TYPE "LBP_typeNCVariableTokenDateAndTime"
TITLE = LBP_ReadVar and LBP_WriteVar Interface / Interface LBP_ReadVar et LBP_WriteVar
// User Data Type for LBP_ReadVar[FB2] and LBP_WriteVar[FB3] Parameters / Type de données utilisateur pour les paramètres LBP_ReadVar[FB2] et LBP_WriteVar[FB3]
   STRUCT
      token : "LBP_typeNCVariableToken";   // User Data Type for LBP_ReadVar[FB2] and LBP_WriteVar[FB3] Input Parameter Addrx / Type de données utilisateur pour les paramètres d'entrée Addrx LBP_ReadVar[FB2] et LBP_WriteVar[FB3]
      value : Date_And_Time;   // Data Type for LBP_ReadVar[FB2] and LBP_WriteVar[FB3] InOut Parameter SDx / Type de données pour les paramètres E/S SDx LBP_ReadVar[FB2] et LBP_WriteVar[FB3]
   END_STRUCT;
END_TYPE

TYPE "LBP_typeNCVariableTokenInt"
TITLE = LBP_ReadVar and LBP_WriteVar Interface / Interface LBP_ReadVar et LBP_WriteVar
// User Data Type for LBP_ReadVar[FB2] and LBP_WriteVar[FB3] Parameters / Type de données utilisateur pour les paramètres LBP_ReadVar[FB2] et LBP_WriteVar[FB3]
   STRUCT
      token : "LBP_typeNCVariableToken";   // User Data Type for LBP_ReadVar[FB2] and LBP_WriteVar[FB3] Input Parameter Addrx / Type de données utilisateur pour les paramètres d'entrée Addrx LBP_ReadVar[FB2] et LBP_WriteVar[FB3]
      value : Int;   // Data Type for LBP_ReadVar[FB2] and LBP_WriteVar[FB3] InOut Parameter SDx / Type de données pour les paramètres E/S SDx LBP_ReadVar[FB2] et LBP_WriteVar[FB3]
   END_STRUCT;
END_TYPE

TYPE "LBP_typeNCVariableTokenLReal"
TITLE = LBP_ReadVar and LBP_WriteVar Interface / Interface LBP_ReadVar et LBP_WriteVar
// User Data Type for LBP_ReadVar[FB2] and LBP_WriteVar[FB3] Parameters / Type de données utilisateur pour les paramètres LBP_ReadVar[FB2] et LBP_WriteVar[FB3]
   STRUCT
      token : "LBP_typeNCVariableToken";   // User Data Type for LBP_ReadVar[FB2] and LBP_WriteVar[FB3] Input Parameter Addrx / Type de données utilisateur pour les paramètres d'entrée Addrx LBP_ReadVar[FB2] et LBP_WriteVar[FB3]
      value : LReal;   // Data Type for LBP_ReadVar[FB2] and LBP_WriteVar[FB3] InOut Parameter SDx / Type de données pour les paramètres E/S SDx LBP_ReadVar[FB2] et LBP_WriteVar[FB3]
   END_STRUCT;
END_TYPE

TYPE "LBP_typeNCVariableTokenReal"
TITLE = LBP_ReadVar and LBP_WriteVar Interface / Interface LBP_ReadVar et LBP_WriteVar
// User Data Type for LBP_ReadVar[FB2] and LBP_WriteVar[FB3] Parameters / Type de données utilisateur pour les paramètres LBP_ReadVar[FB2] et LBP_WriteVar[FB3]
   STRUCT
      token : "LBP_typeNCVariableToken";   // User Data Type for LBP_ReadVar[FB2] and LBP_WriteVar[FB3] Input Parameter Addrx / Type de données utilisateur pour les paramètres d'entrée Addrx LBP_ReadVar[FB2] et LBP_WriteVar[FB3]
      value : Real;   // Data Type for LBP_ReadVar[FB2] and LBP_WriteVar[FB3] InOut Parameter SDx / Type de données pour les paramètres E/S SDx LBP_ReadVar[FB2] et LBP_WriteVar[FB3]
   END_STRUCT;
END_TYPE

TYPE "LBP_typeNCVariableTokenSInt"
TITLE = LBP_ReadVar and LBP_WriteVar Interface / Interface LBP_ReadVar et LBP_WriteVar
// User Data Type for LBP_ReadVar[FB2] and LBP_WriteVar[FB3] Parameters / Type de données utilisateur pour les paramètres LBP_ReadVar[FB2] et LBP_WriteVar[FB3]
   STRUCT
      token : "LBP_typeNCVariableToken";   // User Data Type for LBP_ReadVar[FB2] and LBP_WriteVar[FB3] Input Parameter Addrx / Type de données utilisateur pour les paramètres d'entrée Addrx LBP_ReadVar[FB2] et LBP_WriteVar[FB3]
      value : SInt;   // Data Type for LBP_ReadVar[FB2] and LBP_WriteVar[FB3] InOut Parameter SDx / Type de données pour les paramètres E/S SDx LBP_ReadVar[FB2] et LBP_WriteVar[FB3]
   END_STRUCT;
END_TYPE

TYPE "LBP_typeNCVariableTokenString"
TITLE = LBP_ReadVar and LBP_WriteVar Interface / Interface LBP_ReadVar et LBP_WriteVar
// User Data Type for LBP_ReadVar[FB2] and LBP_WriteVar[FB3] Parameters / Type de données utilisateur pour les paramètres LBP_ReadVar[FB2] et LBP_WriteVar[FB3]
   STRUCT
      token : "LBP_typeNCVariableToken";   // User Data Type for LBP_ReadVar[FB2] and LBP_WriteVar[FB3] Input Parameter Addrx / Type de données utilisateur pour les paramètres d'entrée Addrx LBP_ReadVar[FB2] et LBP_WriteVar[FB3]
      value : String;   // Data Type for LBP_ReadVar[FB2] and LBP_WriteVar[FB3] InOut Parameter SDx / Type de données pour les paramètres E/S SDx LBP_ReadVar[FB2] et LBP_WriteVar[FB3]
   END_STRUCT;
END_TYPE

TYPE "LBP_typeNCVariableTokenUDInt"
TITLE = LBP_ReadVar and LBP_WriteVar Interface / Interface LBP_ReadVar et LBP_WriteVar
// User Data Type for LBP_ReadVar[FB2] and LBP_WriteVar[FB3] Parameters / Type de données utilisateur pour les paramètres LBP_ReadVar[FB2] et LBP_WriteVar[FB3]
   STRUCT
      token : "LBP_typeNCVariableToken";   // User Data Type for LBP_ReadVar[FB2] and LBP_WriteVar[FB3] Input Parameter Addrx / Type de données utilisateur pour les paramètres d'entrée Addrx LBP_ReadVar[FB2] et LBP_WriteVar[FB3]
      value : UDInt;   // Data Type for LBP_ReadVar[FB2] and LBP_WriteVar[FB3] InOut Parameter SDx / Type de données pour les paramètres E/S SDx LBP_ReadVar[FB2] et LBP_WriteVar[FB3]
   END_STRUCT;
END_TYPE

TYPE "LBP_typeNCVariableTokenUInt"
TITLE = LBP_ReadVar and LBP_WriteVar Interface / Interface LBP_ReadVar et LBP_WriteVar
// User Data Type for LBP_ReadVar[FB2] and LBP_WriteVar[FB3] Parameters / Type de données utilisateur pour les paramètres LBP_ReadVar[FB2] et LBP_WriteVar[FB3]
   STRUCT
      token : "LBP_typeNCVariableToken";   // User Data Type for LBP_ReadVar[FB2] and LBP_WriteVar[FB3] Input Parameter Addrx / Type de données utilisateur pour les paramètres d'entrée Addrx LBP_ReadVar[FB2] et LBP_WriteVar[FB3]
      value : UInt;   // Data Type for LBP_ReadVar[FB2] and LBP_WriteVar[FB3] InOut Parameter SDx / Type de données pour les paramètres E/S SDx LBP_ReadVar[FB2] et LBP_WriteVar[FB3]
   END_STRUCT;
END_TYPE

TYPE "LBP_typeNCVariableTokenUSInt"
TITLE = LBP_ReadVar and LBP_WriteVar Interface / Interface LBP_ReadVar et LBP_WriteVar
// User Data Type for LBP_ReadVar[FB2] and LBP_WriteVar[FB3] Parameters / Type de données utilisateur pour les paramètres LBP_ReadVar[FB2] et LBP_WriteVar[FB3]
   STRUCT
      token : "LBP_typeNCVariableToken";   // User Data Type for LBP_ReadVar[FB2] and LBP_WriteVar[FB3] Input Parameter Addrx / Type de données utilisateur pour les paramètres d'entrée Addrx LBP_ReadVar[FB2] et LBP_WriteVar[FB3]
      value : USInt;   // Data Type for LBP_ReadVar[FB2] and LBP_WriteVar[FB3] InOut Parameter SDx / Type de données pour les paramètres E/S SDx LBP_ReadVar[FB2] et LBP_WriteVar[FB3]
   END_STRUCT;
END_TYPE

DATA_BLOCK "DB_WAF"   // DB12
{ S7_Optimized_Access := 'TRUE' }
// stored: MemoryReserve 100
   VAR
      bTest : Array[0..63] of Bool;
      bSpy : Array[0..63] of Bool;
      Sonplas : Struct
         OperateInOutCollision : Bool;
      END_STRUCT;
      BwLoader : Struct
         Safe : Bool;
         Auto : Bool;
      END_STRUCT;
      CtrlInEnable : Bool := true;
      CtrlOutEnable : Bool := true;
      CtrlBwEnable : Bool := true;
      U2States : Byte;
      ResetPartPosition : Bool;
      HMI_Pos : Bool;
      PLC_Pos : Bool;
      NewTag : Bool;
      NewTag_1 : Bool;
   END_VAR
BEGIN
END_DATA_BLOCK

DATA_BLOCK "DB_HMICmd"   // DB86
{ S7_Optimized_Access := 'TRUE' }
// stored: MemoryReserve 100
   VAR
      IntGateCloseReq : Bool;
      IntGateOpenReq : Bool;
      ExtGateCloseReq : Bool;
      ExtGateOpenReq : Bool;
      IntGateCloseCmd : Bool;
      IntGateOpenCmd : Bool;
      ExtGateCloseCmd : Bool;
      ExtGateOpenCmd : Bool;
      BlowingCmd : Bool;
   END_VAR
BEGIN
END_DATA_BLOCK

DATA_BLOCK "DB_HMISetting"   // DB1306
{ S7_Optimized_Access := 'FALSE' }
AUTHOR : DAT
NAME : IHM_SETT
// stored: AutoNumber false
   VAR RETAIN
      GasAssistSetPoint : Real;
      CoolingVentilatorSetpoint : Real;   // @Precision:0 @Unit:% @Min:0 @Max:100
      TemperatureCoolingSetpoint : Real;   // @Precision:1 @Unit:°C @Min:0 @Max:50
      BlowingSetpoint : Real;   // @Precision:0 @Unit:ms @Min:0 @Max:500
      WorkingMode : Struct
         EmptyingReq : Bool;
      END_STRUCT;
      Sonplas : Struct
         LimitMax : Real;
         LimitCtrlMax : Real;
         LimitCtrlMin : Real;
         LimitMin : Real;
         CorrectionMax : Real;
         CorrectionMin : Real;
      END_STRUCT;
      LockDoorReq : Bool;
      UnlockDoorReq : Bool;
      StartAutoReq : Bool;
      StopAutoReq : Bool;
      Shuttle1Enable : Bool;
      Shuttle2Enable : Bool;
   END_VAR
BEGIN
END_DATA_BLOCK

DATA_BLOCK "DB_HMIStatus"   // DB95
{ S7_Optimized_Access := 'TRUE' }
// stored: MemoryReserve 100
   VAR
      WarmUpOn : Bool := FALSE;
      WarmUpTime : Real := 30.0;
      KeyLaserOn : Bool := TRUE;
      Shutter_laser_closed : Bool := FALSE;
      Sonplas : Struct
         LastMeasure : Real;
         CurrentCorrection : Real;
         CouplerOk : Bool;
         Ready : Bool;
      END_STRUCT;
   END_VAR
BEGIN
END_DATA_BLOCK

DATA_BLOCK "DB_MachineOptions"   // DB1300
{ S7_Optimized_Access := 'FALSE'; DB_Accessible_From_OPC_UA := 'FALSE' }
// stored: AutoNumber false, DBAccessibleFromOPCUA false, DBAccessibleFromWebserver false
   VAR RETAIN
      UPSPresent : Bool;
      Fixture : Struct
         Passive_Open : Bool;
      END_STRUCT;
      Mach_MONO_DUO : Bool;
      Chiller : Struct
         Termotek : Bool := TRUE;
         SMC : Bool := FALSE;
      END_STRUCT;
   END_VAR
BEGIN
END_DATA_BLOCK

DATA_BLOCK "DB_PLC_ISO_IHM"   // DB1302
{ S7_Optimized_Access := 'FALSE' }
AUTHOR : SAN
FAMILY : DPR
NAME : HMI
// stored: AutoNumber false
   VAR RETAIN
      WarmUpOn : Bool := FALSE;   // Moved to DB_HMI_Status
      KeyLaserOn : Bool := TRUE;   // Moved to DB_HMI_Status
      KeySaveParameters : Bool := FALSE;   // Not used
      bStopAfterEmptying : Bool := FALSE;   // A VOIR SI ENCORE UTILE
      Chan1_running : Bool := TRUE;   // Moved to DB_HMI_Status
      Chan2_running : Bool := FALSE;   // Moved to DB_HMI_Status
      Chan3_running : Bool := FALSE;   // Moved to DB_HMI_Status
      Chan4_running : Bool := FALSE;   // Moved to DB_HMI_Status
      StopAtNextReq { S7_SetPoint := 'True'} : Bool := FALSE;   // Moved to DB_HMI_Status
      AllChanStop : Bool := FALSE;   // Moved to DB_HMI_Status
      LoaderAutomaticMode : Bool := FALSE;   // A VOIR SI ENCORE UTILE
      LoaderManualMode : Bool := TRUE;   // A VOIR SI ENCORE UTILE
      NoCameraPresent : Bool := FALSE;   // Not used
      PremeasureZexists : Bool := FALSE;   // Not used
      PremeasureCexists : Bool := FALSE;   // Not used
      PLCFunctNotFinished : Bool := FALSE;   // Not used
      StartChangePart_station1 : Bool := FALSE;   // A VOIR SI ENCORE UTILE
      StartCheckPart_fixture1 : Bool := FALSE;   // A VOIR SI ENCORE UTILE
      Loader1PartLoad : Bool := FALSE;   // A VOIR SI ENCORE UTILE
      Loader1PartUnload : Bool := FALSE;   // A VOIR SI ENCORE UTILE
      Loader1ShiftLoad : Bool := FALSE;   // A VOIR SI ENCORE UTILE
      Loader1ShiftUnload : Bool := FALSE;   // A VOIR SI ENCORE UTILE
      Loader1LoadOpened : Bool := TRUE;   // A VOIR SI ENCORE UTILE
      Loader1UnloadOpened : Bool := TRUE;   // A VOIR SI ENCORE UTILE
      PartOnFixture1 : Bool := FALSE;   // A VOIR SI ENCORE UTILE
      MasterOnFixture1 : Bool := FALSE;   // A VOIR SI ENCORE UTILE
      StartChangePart_station2 : Bool := FALSE;   // A VOIR SI ENCORE UTILE
      StartCheckPart_fixture2 : Bool := FALSE;   // A VOIR SI ENCORE UTILE
      Loader2PartLoad : Bool := FALSE;   // A VOIR SI ENCORE UTILE
      Loader2PartUnload : Bool := FALSE;   // A VOIR SI ENCORE UTILE
      Loader2ShiftLoad : Bool := FALSE;   // A VOIR SI ENCORE UTILE
      Loader2ShiftUnload : Bool := FALSE;   // A VOIR SI ENCORE UTILE
      Loader2LoadOpened : Bool := FALSE;   // A VOIR SI ENCORE UTILE
      Loader2UnloadOpened : Bool := FALSE;   // A VOIR SI ENCORE UTILE
      PartOnFixture2 : Bool := FALSE;   // A VOIR SI ENCORE UTILE
      MasterOnFixture2 : Bool := FALSE;   // A VOIR SI ENCORE UTILE
      StartChangePart_station3 : Bool := FALSE;   // A VOIR SI ENCORE UTILE
      StartCheckPart_fixture3 : Bool := FALSE;   // A VOIR SI ENCORE UTILE
      Loader3PartLoad : Bool := FALSE;   // A VOIR SI ENCORE UTILE
      Loader3PartUnload : Bool := FALSE;   // A VOIR SI ENCORE UTILE
      Loader3ShiftLoad : Bool := FALSE;   // A VOIR SI ENCORE UTILE
      Loader3ShiftUnload : Bool := FALSE;   // A VOIR SI ENCORE UTILE
      Loader3LoadOpened : Bool := FALSE;   // A VOIR SI ENCORE UTILE
      Loader3UnloadOpened : Bool := FALSE;   // A VOIR SI ENCORE UTILE
      PartOnFixture3 : Bool := FALSE;   // A VOIR SI ENCORE UTILE
      MasterOnFixture3 : Bool := FALSE;   // A VOIR SI ENCORE UTILE
      Part_KO_go_outside_mach : Bool := TRUE;   // Not used
      MasterOnMachine : Bool := FALSE;   // Not used
      Part_position_1 : Bool := FALSE;   // A VOIR COMMENT GERER AVEC TRACABILITY
      Part_position_2 : Bool := FALSE;   // A VOIR COMMENT GERER AVEC TRACABILITY
      Part_position_3 : Bool := FALSE;   // A VOIR COMMENT GERER AVEC TRACABILITY
      Part_position_4 : Bool := FALSE;   // A VOIR COMMENT GERER AVEC TRACABILITY
      Part_position_5 : Bool := FALSE;   // A VOIR COMMENT GERER AVEC TRACABILITY
      Part_position_6 : Bool := FALSE;   // A VOIR COMMENT GERER AVEC TRACABILITY
      Part_position_7 : Bool := FALSE;   // A VOIR COMMENT GERER AVEC TRACABILITY
      Part_position_8 : Bool := FALSE;   // A VOIR COMMENT GERER AVEC TRACABILITY
      Part_position_9 : Bool := FALSE;   // A VOIR COMMENT GERER AVEC TRACABILITY
      Part_position_10 : Bool := FALSE;   // A VOIR COMMENT GERER AVEC TRACABILITY
      Part_position_11 : Bool := FALSE;   // A VOIR COMMENT GERER AVEC TRACABILITY
      Part_position_12 : Bool := FALSE;   // A VOIR COMMENT GERER AVEC TRACABILITY
      Part_position_13 : Bool := FALSE;   // A VOIR COMMENT GERER AVEC TRACABILITY
      Part_position_14 : Bool := FALSE;   // A VOIR COMMENT GERER AVEC TRACABILITY
      Part_position_15 : Bool := FALSE;   // A VOIR COMMENT GERER AVEC TRACABILITY
      Part_position_16 : Bool := FALSE;   // A VOIR COMMENT GERER AVEC TRACABILITY
      WarmUpTime : Int := 30;   // Moved to DB_HMI_Status
      Stop_For_BackWall_Wear_1 : Bool := FALSE;   // Moved to DB_HMI_Status
      Stop_For_BackWall_Wear_2 : Bool := FALSE;   // Moved to DB_HMI_Status
      Cleaning_Station_1 : Bool := FALSE;   // Moved to DB_HMI_Status
      Cleaning_Station_2 : Bool := FALSE;   // Moved to DB_HMI_Status
      Cleaning_Backwall_1 : Bool := FALSE;   // Moved to DB_HMI_Status
      Cleaning_Backwall_2 : Bool := FALSE;   // Moved to DB_HMI_Status
      Shutter_laser_closed : Bool := FALSE;   // Moved to DB_HMI_Status
      Pressure_Stop_Machine : Bool := FALSE;   // Moved to DB_HMI_Status
      Set_Bad_Part_On_Fixture : Bool := FALSE;   // Moved to DB_HMI_Status
      Reserve12 : Bool := FALSE;   // Not used
      Reserve13 : Bool := FALSE;   // Not used
      Reserve14 : Bool := FALSE;   // Not used
      Reserve15 : Bool := FALSE;   // Not used
      SemiAuto_RunEmpty : Bool := FALSE;   // A VOIR SI ENCORE UTILE
      "SemiAuto_Unload_C-Fixture" : Bool := FALSE;   // A VOIR SI ENCORE UTILE
      Reserve18 : Bool := FALSE;   // Not used
      Cnt_Washing_Loader_1 : Int := 1;   // A VOIR SI ENCORE UTILE
      Cnt_Washing_Loader_2 : Int := 0;   // A VOIR SI ENCORE UTILE
      Cnt_Part_Backwall_1 : Int := 16;   // Moved to DB_HMI_Status
      Cnt_Part_Backwall_2 : Int := 0;   // Moved to DB_HMI_Status
      Cnt_Part_Wash_Backwall_1 : Int := 26;   // Moved to DB_HMI_Status
      Cnt_Part_Wash_Backwall_2 : Int := 0;   // Moved to DB_HMI_Status
      Cnt_Part_Blow_Fixture_1 : Int;   // Moved to DB_HMI_Status
      Cnt_Part_Blow_Fixture_2 : Int;   // Moved to DB_HMI_Status
      Setpoint_laser_air_process : Real;   // Not used
      StopMachine : Bool;   // Not used
      BadPartOnFixture : Bool;   // Not used
   END_VAR
BEGIN
END_DATA_BLOCK

DATA_BLOCK "DB_LoaderOptions"   // DB1305
{ S7_Optimized_Access := 'TRUE' }
AUTHOR : SAN
// stored: AutoNumber false, IsRetainMemResEnabled true, MemoryReserve 20, RetainMemoryReserve 20
   VAR RETAIN
      ExtLoadUnload : Struct
         SeparatePos : Bool;
         CommonPos : Bool;
         Disabled : Bool;
      END_STRUCT;
      Blowing : Struct
         Inside : Bool;
         NearSas : Bool;
         Disabled : Bool;
      END_STRUCT;
      Washing : Struct
         Enabled : Bool;
         Disabled : Bool;
      END_STRUCT;
      PartControl : Struct
         Individual : Bool;
         Common : Bool;
         Disabled : Bool;
         AnalogMeasure : Bool;
         DigitalMeasure : Bool;
      END_STRUCT;
   END_VAR
   VAR
      Stop_Restart : Struct
         BasicVersion : Bool;
      END_STRUCT;
      IntLoadUnload : Struct
         SeparatePos : Bool;
         CommonPos : Bool;
      END_STRUCT;
      BwLoadUnload : Struct
         SeparatePos : Bool;
         CommonPos : Bool;
      END_STRUCT;
      BwControl : Struct
         UndrilledDrilledCtrlSeparate : Bool;
         UndrilledDrilledCtrlCommon : Bool;
         Disabled : Bool;
      END_STRUCT;
      ActPartControlIn : Struct
         Stop : Bool := TRUE;
      END_STRUCT;
      ActPartControlOut : Struct
         Stop : Bool := TRUE;
      END_STRUCT;
      ActBwControlIn : Struct
         Stop : Bool := TRUE;
      END_STRUCT;
      Fixture : Struct
         UnloadingDisabled : Bool;
         LoadingDisabled : Bool;
         BlowingDisabled : Bool;
         ReleaseDisabled : Bool;
         V_InitDisabled : Bool;
         W_InitDisabled : Bool;
      END_STRUCT;
   END_VAR
BEGIN
END_DATA_BLOCK

DATA_BLOCK "DB_ActiveAlarms"   // DB115
{ S7_Optimized_Access := 'TRUE' }
// stored: MemoryReserve 100
   VAR
      NumberOfActiveAlarms : DInt;
      ActiveAlarms : Array[0..50] of "UDT_Alarms";
      Update { S7_SetPoint := 'True'} : Byte;   // A modifier lors d'un Acknowledge
   END_VAR
BEGIN
END_DATA_BLOCK

DATA_BLOCK "DB_FormatMsg"   // DB18
{ S7_Optimized_Access := 'TRUE' }
// stored: MemoryReserve 100
   VAR
      Msg : Array[0..863] of "UDT_FormatMsg";
   END_VAR
BEGIN
END_DATA_BLOCK

DATA_BLOCK "DB_AxisPosMachineNC"   // DB82
{ S7_Optimized_Access := 'TRUE' }
// stored: MemoryReserve 100
   VAR
      Axis_X : Struct
         Load : LReal := 249.3;
         Unload : LReal := 324.5;
         Blowing : LReal := 287.3;
      END_STRUCT;
      Axis_Y : Struct
         Load : LReal := 55.02;
         Unload : LReal := 55.02;
         Blowing : LReal := 55.02;
      END_STRUCT;
      Axis_B : Struct
         Load : LReal := 0.0;
         Unload : LReal := 0.0;
         Blowing : LReal := 0.0;
      END_STRUCT;
      Axis_ZM : Struct
         Safe : Real := 145.0;
      END_STRUCT;
      Axis_ZL : Struct
         Safe : Real := 14.0;
      END_STRUCT;
   END_VAR
BEGIN
END_DATA_BLOCK

DATA_BLOCK "DB_AxisPosMachinePLC"   // DB103
{ S7_Optimized_Access := 'TRUE' }
// stored: AutoNumber false, MemoryReserve 100
   VAR
      Axis_U1 : Struct
         ExtLoadUnloadAuto : LReal := -3370.0;
         ExtLoadUnloadManu : LReal := -3365.0;
         PartControl : LReal := -3257.0;
         BwLoad : LReal := -1886.83;
         BwUnLoad : LReal := -1962.83;
         BwControl : LReal := -1775.0;
         IntLoadUnload : LReal := -0.2;
         ExtGateExt : LReal := -1164.0;
         IntGateExt : LReal := -857.0;
         ExtGateInt : LReal := -809.0;
         IntGateInt : LReal := -502.0;
         Sas : LReal := -833.0;
         Blowing : LReal := 36.0;
         IntLoadUnloadOP : LReal := 76.0;
      END_STRUCT;
      Axis_U2 : Struct
         ExtLoadUnloadAuto : LReal := -3370.0;
         ExtLoadUnloadManu : LReal := -3365.0;
         PartControl : LReal := -3257.0;
         BwLoad : LReal := -1886.78;
         BwUnLoad : LReal := -1962.78;
         BwControl : LReal := -1775.0;
         IntLoadUnload : LReal := -0.11;
         ExtGateExt : LReal := -1164.0;
         IntGateExt { ExternalAccessible := 'False'; ExternalVisible := 'False'; ExternalWritable := 'False'} : LReal := -857.0;
         ExtGateInt : LReal := -809.0;
         IntGateInt : LReal := -502.0;
         Sas : LReal := -833.0;
         Blowing : LReal := 36.0;
         IntLoadUnloadOP : LReal := 76.0;
      END_STRUCT;
      Axis_V : Struct
         Shuttle_1 : Struct
            LoadUnload : LReal := 17.95;
            Blowing : LReal := 17.95;
         END_STRUCT;
         Shuttle_2 : Struct
            LoadUnload : LReal := -0.48;
            Blowing : LReal := -0.48;
         END_STRUCT;
         Safe : LReal := -0.48;
         Fixture : Struct
            Safe : LReal := 40.0;
            Load : LReal := 192.62;   // 193.52
            Unload : LReal := 192.62;   // 193.52
            Blowing : LReal := 192.62;   // 193.52
         END_STRUCT;
      END_STRUCT;
      Axis_W : Struct
         Shuttle_1 : Struct
            Approach : LReal := -17.61;
            LoadUnload : LReal := -19.61;
            Blowing : LReal := -5.0;
         END_STRUCT;
         Shuttle_2 : Struct
            Approach : LReal := -17.81;
            LoadUnload : LReal := -19.81;
            Blowing : LReal := -5.0;
         END_STRUCT;
         Safe : LReal := 28.5;
         Fixture : Struct
            Safe : LReal := 28.5;
            Load : LReal := -0.8;
            Blowing : LReal := 15.0;
            Unload : LReal := -0.9;
            Approach : LReal := 2.0;
         END_STRUCT;
      END_STRUCT;
   END_VAR
BEGIN
END_DATA_BLOCK

DATA_BLOCK "DB_DataFinalPart"   // DB700
{ S7_Optimized_Access := 'TRUE' }
// stored: AutoNumber false, MemoryReserve 100
   VAR
      FinalPart : Array[0..100] of "UDT_Tracability";
   END_VAR
BEGIN
END_DATA_BLOCK

DATA_BLOCK "DB_DataPositions"   // DB701
{ S7_Optimized_Access := 'TRUE' }
// stored: AutoNumber false, MemoryReserve 100
   VAR
      Position : Array[0..52] of "UDT_Tracability";
   END_VAR
BEGIN
END_DATA_BLOCK

DATA_BLOCK "DB_OPC_Buttons"   // DB92
{ S7_Optimized_Access := 'TRUE' }
// stored: MemoryReserve 100
   VAR
      Door : "UDT_OPC_Button";
      Empty : "UDT_OPC_Button";
      Start : "UDT_OPC_Button";
      Stop : "UDT_OPC_Button";
      Powermeter { S7_SetPoint := 'True'} : "UDT_OPC_Button";
      GasAssist { S7_SetPoint := 'True'} : "UDT_OPC_Button";
      GripperUndrilledClamp : Struct
         Close : "UDT_OPC_Button";
         Open { S7_SetPoint := 'True'} : "UDT_OPC_Button";
         IsClosed { S7_SetPoint := 'True'} : Bool;
         IsOpened { S7_SetPoint := 'True'} : Bool;
      END_STRUCT;
      GripperDrilledClamp : Struct
         Close : "UDT_OPC_Button";
         Open { S7_SetPoint := 'True'} : "UDT_OPC_Button";
         IsClosed { S7_SetPoint := 'True'} : Bool;
         IsOpened { S7_SetPoint := 'True'} : Bool;
      END_STRUCT;
      SITestStop { S7_SetPoint := 'True'} : "UDT_OPC_Button";
      FixtureClamp { S7_SetPoint := 'True'} : "UDT_OPC_Button";
      FixtureVacuum { S7_SetPoint := 'True'} : "UDT_OPC_Button";
      Aspiration { S7_SetPoint := 'True'} : "UDT_OPC_Button";
      LoaderAuto { S7_SetPoint := 'True'} : "UDT_OPC_Button";
      LoaderSemiAuto { S7_SetPoint := 'True'} : "UDT_OPC_Button";
      Backlight { S7_SetPoint := 'True'} : "UDT_OPC_Button";
      ObservationCamera { S7_SetPoint := 'True'} : "UDT_OPC_Button";
      MainDoor { S7_SetPoint := 'True'} : "UDT_OPC_Button";
      WarmUp { S7_SetPoint := 'True'} : "UDT_OPC_Button";
      MachineLight { S7_SetPoint := 'True'} : "UDT_OPC_Button";
   END_VAR
BEGIN
END_DATA_BLOCK

DATA_BLOCK "DB_OPC_Axis"   // DB102
{ S7_Optimized_Access := 'TRUE' }
// stored: MemoryReserve 100
   VAR
      ActualValues : Struct
         NumberOfAxes { S7_SetPoint := 'True'} : DInt;
         Axes : Array[0..100] of "UDT_OPC_ActualValuesAxis";
      END_STRUCT;
      TaughtPositions : Struct
         NumberOfItems { S7_SetPoint := 'True'} : DInt;
         Items : Array[0..100] of "UDT_OPC_TaughtPositionsItems";
      END_STRUCT;
      Teach : Struct
         Buttons : Struct
            Teach : "UDT_OPCButtons";
         END_STRUCT;
         Parameters : Struct
            AxisId : DInt;
            PositionId : DInt;
         END_STRUCT;
         Current : Struct
            ActualPosition : LReal;
            TaughtPosition : LReal;
         END_STRUCT;
      END_STRUCT;
   END_VAR
BEGIN
END_DATA_BLOCK

DATA_BLOCK "DB_OPC_Machine"   // DB15
{ S7_Optimized_Access := 'TRUE' }
// stored: MemoryReserve 100
   VAR
      Parts : Struct
         Out : Struct
            Station1 : Struct
               LoaderDrilled : SInt;
               LoaderUndrilled : SInt;
               ShuttleDrilled : SInt;
               ShuttleUndrilled : SInt;
               WorkClamp : SInt;
            END_STRUCT;
         END_STRUCT;
      END_STRUCT;
      State : Struct
         Current : Struct
            CanLockDoor : Bool;
            CanUnlockDoor : Bool;
            CncMode : Byte;
            LoadingMode : Byte;
            IsDoorLocked : Bool;
            IsEmptying : Bool;
            IsInitialized : Bool;
            IsRunning : Bool;
            MachineOverride : Byte;
         END_STRUCT;
         Requests : Struct
            LoadingMode : Struct
               RequestChangeMode : Bool;
               TargetMode : Byte;
            END_STRUCT;
            RequestLockDoor : Bool;
            RequestStartAuto : Bool;
            RequestStartEmptying : Bool;
            RequestStopAuto : Bool;
            RequestStopEmptying : Bool;
            RequestUnlockDoor : Bool;
         END_STRUCT;
      END_STRUCT;
   END_VAR
   VAR RETAIN
      Parameters : Struct
         GasAssistSetPoint : Real;
         CoolingVentilatorSetpoint : Real;
         TemperatureCoolingSetpoint : Real;
         BlowingSetpoint : Real;
         Shuttle1Enable : "UDT_BoolEnable";
         Shuttle2Enable { S7_SetPoint := 'True'} : "UDT_BoolEnable";
         ConsecutiveBwIn { S7_SetPoint := 'True'} : Int;
         Sequence : Struct
            Shuttle1 : Struct
               Main : Int;
               ShuttleInt : Int;
               ShuttleExt : Int;
               ControlIn : Int;
               ControlOut : Int;
               Blowing : Int;
               IntLoadUnload : Int;
               ExtLoadUnload : Int;
               BwLoadUnload : Int;
               BwControlIn : Int;
               ActControlIn : Int;
               ActControlOut : Int;
               ActBwControlIn : Int;
            END_STRUCT;
            Shuttle2 : Struct
               Main : Int;
               ShuttleInt : Int;
               ShuttleExt : Int;
               ControlIn : Int;
               ControlOut : Int;
               Blowing : Int;
               IntLoadUnload : Int;
               ExtLoadUnload : Int;
               BwLoadUnload : Int;
               BwControlIn : Int;
               ActControlIn : Int;
               ActControlOut : Int;
               ActBwControlIn : Int;
            END_STRUCT;
            Fixture : Struct
               Blowing : Int;
               Loading : Int;
               Unloading : Int;
               V_Init : Int;
               W_Init : Int;
            END_STRUCT;
         END_STRUCT;
         Presence : Struct
            Shuttle1UndrilledPart : Bool;
            Shuttle1UndrilledBw : Bool;
            Shuttle1DrilledPart : Bool;
            Shuttle1DrilledBw : Bool;
            Shuttle2UndrilledPart : Bool;
            Shuttle2UndrilledBw : Bool;
            Shuttle2DrilledPart : Bool;
            Shuttle2DrilledBw : Bool;
            GripperUndrilledPart : Bool;
            GripperUndrilledBw : Bool;
            GripperDrilledPart : Bool;
            GripperDrilledBw : Bool;
            FixtureUndrilledPart : Bool;
            FixtureUndrilledBw : Bool;
            FixtureDrilledPart : Bool;
            FixtureDrilledBw : Bool;
         END_STRUCT;
      END_STRUCT;
   END_VAR
BEGIN
END_DATA_BLOCK

DATA_BLOCK "DB_OPC_Alarms"   // DB117
{ S7_Optimized_Access := 'TRUE' }
// stored: MemoryReserve 100
   VAR
      NumberOfActiveAlarms : DInt;
      ActiveAlarms : Array[0..50] of "UDT_Alarms";
      Update { S7_SetPoint := 'True'} : Byte;   // A modifier lors d'un Acknowledge
   END_VAR
BEGIN
END_DATA_BLOCK

DATA_BLOCK "DB_BwLoaderExchange"   // DB101
{ S7_Optimized_Access := 'TRUE' }
// stored: MemoryReserve 100
   VAR
      Inputs : Struct
         LifeFlag : Int;
         JobDone : Bool;
         LockShuttle : Bool;
         DataSend : Int;
         DataReceive : Int;
         NoEmergencyStopAtBwLoader : Bool;
         SafetyDoorsClosedAtBwLoader : Bool;
         BwInErrorState : Int;
         UndrilledPartControl : Bool;
         DrilledPartControl : Bool;
         BackwallControl : Bool;
         BwLoaderInSafePos : Bool;
      END_STRUCT;
      Outputs : Struct
         LifeFlag : Int;
         LoaderRequest : Bool;
         LockShuttle : Bool;
         DataSend : Int;
         DataReceive : Int;
         NoEmergencyStopAtFemto : Bool;
         SafetyDoorsClosedAtFemto : Bool;
         FemtoInErrorState : Int;
         AutoMode : Bool;
         JogMode : Bool;
         GotoSafePos : Bool;
         Emptying : Bool;
         BW_CtrlInProgress : Bool;
      END_STRUCT;
   END_VAR
BEGIN
END_DATA_BLOCK

DATA_BLOCK "DB_OPC_RealTime"   // DB104
{ S7_Optimized_Access := 'TRUE' }
// stored: MemoryReserve 100
   VAR
      GripperUndrilledClampOpen : Bool;   // Test
      GripperUndrilledClampClosed : Bool;   // Test
      FixturePosition : Real;   // Test
      X_AxisBrakePressCtrl : Bool;   // Digital Input
      Y_AxisBrakePressCtrl : Bool;   // Digital Input
      BreakerCtrl : Bool;   // Digital Input
      CabinetTemperatureCtrl : Bool;   // Digital Input
      UpsPowerFailure : Bool;   // Digital Input
      AirPressureCtrl : Bool;   // Digital Input
      ShutterClosed : Bool;   // Digital Input
      AirDryerOK : Bool;   // Digital Input
      UPS_BatteryOK : Bool;   // Digital Input
      FrontDoorClosed : Bool;   // Digital Input
      InfeedReadyOkStart : Bool;   // Digital Input
      CoolingOK : Bool;   // Digital Input
      PowerReady : Bool;   // Digital Input
      AlarmI2T : Bool;   // Digital Input
      HeadLaserBusy : Bool;   // Digital Input
      HeadLaserBreaker : Bool;   // Digital Input
      FrontDoorLocked : Bool;   // Digital Input
      UPS_CommonAlarm : Bool;   // Digital Input
      UPS_BatteryLow : Bool;   // Digital Input
      HeadChillerHighPressure : Bool;   // Digital Input
      HeadChillerWaterTemperature : Bool;   // Digital Input
      HeadChillerFlow : Bool;   // Digital Input
      HeadChillerCollectivFault : Bool;   // Digital Input
      HeadChillerWaterLevel : Bool;   // Digital Input
      UpsByPassActive : Bool;   // Digital Input
      HeadChillerAmbiantTemperature : Bool;   // Digital Input
      LoadClampOpened : Bool;   // Digital Input
      LoadClampNotClosedWithPart : Bool;   // Digital Input
      UnloadClampOpened : Bool;   // Digital Input
      UpsFault : Bool;   // Digital Input
      InternalGateLocked : Bool;   // Digital Input
      ExternalGateLocked : Bool;   // Digital Input
      InverterActive : Bool;   // Digital Input
      UnloadClampNotClosedWithPart : Bool;   // Digital Input
      InternalGateOpened : Bool;   // Digital Input
      ExternalGateOpened : Bool;   // Digital Input
      PowerMeterBackCtrl : Bool;   // Digital Input
      PowerMeterFrontCtrl : Bool;   // Digital Input
      HeadChillerCutOff : Bool;   // Digital Input
      HeadChillerTemperature : Bool;   // Digital Input
      ClampingOpenCtrl : Bool;   // Digital Input
      B_AxisBrakeReleasedCtrl : Bool;   // Digital Input
      B_AxisReferencePoint : Bool;   // Digital Input
      SourceChillerHighPressure : Bool;   // Digital Input
      SourceChillerWaterTemperature : Bool;   // Digital Input
      SourceChillerFlow : Bool;   // Digital Input
      SourceChillerCollectivFault : Bool;   // Digital Input
      SourceChillerWaterLevel : Bool;   // Digital Input
      SourceChillerAmbiantTemperature : Bool;   // Digital Input
      SourceChillerCutOff : Bool;   // Digital Input
      SourceChillerTemperature : Bool;   // Digital Input
      OperatingCounter : Bool;   // Digital Output
      GeneralAirValve : Bool;   // Digital Output
      SmartLineDisable : Bool;   // Digital Output
      MachineLight : Bool;   // Digital Output
      MachineLightBack : Bool;   // Digital Output
      LightTowerOrange : Bool;   // Digital Output
      LightTowerRed : Bool;   // Digital Output
      LightTowerBlue : Bool;   // Digital Output
      LightTowerGreen : Bool;   // Digital Output
      LightTowerWhite : Bool;   // Digital Output
      Backlight : Bool;   // Digital Output
      InfeedON : Bool;   // Digital Output
      AxisActivation : Bool;   // Digital Output
      BuzzerActivation : Bool;   // Digital Output
      ElbaronPowerON : Bool;   // Digital Output
      ObservationCameraLight : Bool;   // Digital Output
      LaserExternalDoorOpening : Bool;   // Digital Output
      CoolingStart : Bool;   // Digital Output
      X_AxisBrakeActivation : Bool;   // Digital Output
      Y_AxisBrakeActivation : Bool;   // Digital Output
      AxisB_TeachInClampingPart : Bool;   // Digital Output
      EPO_UPS : Bool;   // Digital Output
      HeadLaserStart : Bool;   // Digital Output
      HeadLaserStop : Bool;   // Digital Output
      Axis2_PowerContactor : Bool;   // Digital Output
      GasAssistOn : Bool;   // Digital Output
      SmartLineReset : Bool;   // Digital Output
      XY_AxisPowerContactor : Bool;   // Digital Output
      LaserAirPressureProcess : Bool;   // Digital Output
      Bus60V_PowerContactor : Bool;   // Digital Output
      LoadClampClosing : Bool;   // Digital Output
      LoadClampOpening : Bool;   // Digital Output
      UnloadClampClosing : Bool;   // Digital Output
      UnloadClampOpening : Bool;   // Digital Output
      ClampingOpening : Bool;   // Digital Output
      ClampingClosing : Bool;   // Digital Output
      B_AxisBrakeRelease : Bool;   // Digital Output
      Suction : Bool;   // Digital Output
      ExternalGateClosing : Bool;   // Digital Output
      ExternalGateOpening : Bool;   // Digital Output
      InternalGateClosing : Bool;   // Digital Output
      InternalGateOpening : Bool;   // Digital Output
      PowerMeterRetract : Bool;   // Digital Output
      PowerMeterAdvance : Bool;   // Digital Output
      Blowing : Bool;   // Digital Output
      LaserPowerMeter : Real;   // Analog Input
      AxisB_ClampingPart : Real;   // Analog Input
      LaserAirPressureProcess_1 : Real;   // Analog Input
      InletAirPressure : Real;   // Analog Input
      AmbiantTemperature : Real;   // Analog Input
      MachineTemperature : Real;   // Analog Input
      Cold_WaterTemperatureInput { ExternalWritable := 'False'} : Real;   // Analog Input
      Cold_WaterTemperatureOutput : Real;   // Analog Input
      X_AxisTemperaturePT1000 : Real;   // Analog Input
      Y_AxisTemperaturePT1000 : Real;   // Analog Input
      X_AxisTemperaturePTC : Real;   // Analog Input
      Y_AxisTemperaturePTC : Real;   // Analog Input
      NozzleOverpressure : Real;   // Analog Input
      OpticalPathOverpressure : Real;   // Analog Input
      LaserHeadOverpressure : Real;   // Analog Input
      ZLAxisOverpressure : Real;   // Analog Input
      XYAxisOverpressure : Real;   // Analog Input
      LeftAspiration : Real;   // Analog Input
      RightAspiration : Real;   // Analog Input
      ClimTemperature : Real;   // Analog Input
      SensorControllerStation1 : Real;   // Analog Input
      CabinetTemperature : Real;   // Analog Input
      NozzleOverpressureSetPoint : Real;   // Analog Output
      VentilatorSetPoint : Real;   // Analog Output
      PropValveClimSetPoint : Real;   // Analog Output
   END_VAR
BEGIN
END_DATA_BLOCK

DATA_BLOCK "DB_OPC_AnalogInputs"   // DB83
{ S7_Optimized_Access := 'TRUE' }
// stored: MemoryReserve 100
   VAR
      NumberOfSignals : Int := 22;
      Parameters : Struct
         Delay : LReal;
         DiffErrorMax : LReal;
         DiffErrorMin : LReal;
         DiffWarnMax : LReal;
         DiffWarnMin : LReal;
         Id : DInt;
         ItemNumber : DInt;
         Offset : LReal := 1.0;
         Gain : LReal;
         Target : LReal;
      END_STRUCT;
      Signals : Array[0..100] of "UDT_OPC_Analog";
      Update { S7_SetPoint := 'True'} : Bool;
   END_VAR
BEGIN
   // Signals[1].DiffErrorMax : Unit:W
   // Signals[3].DiffErrorMax : Unit:bar
   // Signals[4].DiffErrorMax : Unit:°C
   // Signals[5].DiffErrorMax : Unit:°C
   // Signals[6].DiffErrorMax : Unit:°C
   // Signals[7].DiffErrorMax : Unit:°C
   // Signals[8].DiffErrorMax : Unit:°C
   // Signals[9].DiffErrorMax : Unit:°C
   // Signals[10].DiffErrorMax : Unit:°C
   // Signals[13].DiffErrorMax : Unit:bar
   // Signals[14].DiffErrorMax : Unit:bar
   // Signals[15].DiffErrorMax : Unit:bar
   // Signals[16].DiffErrorMax : Unit:bar
   // Signals[17].DiffErrorMax : Unit:bar
   // Signals[18].DiffErrorMax : Unit:mm/s
   // Signals[19].DiffErrorMax : Unit:mm/s
   // Signals[21].DiffErrorMax : Unit:°C
   // Signals[26].DiffErrorMax : Unit:°C
   // Signals[1].DiffErrorMin : Unit:W
   // Signals[3].DiffErrorMin : Unit:bar
   // Signals[4].DiffErrorMin : Unit:°C
   // Signals[5].DiffErrorMin : Unit:°C
   // Signals[6].DiffErrorMin : Unit:°C
   // Signals[7].DiffErrorMin : Unit:°C
   // Signals[8].DiffErrorMin : Unit:°C
   // Signals[9].DiffErrorMin : Unit:°C
   // Signals[10].DiffErrorMin : Unit:°C
   // Signals[13].DiffErrorMin : Unit:bar
   // Signals[14].DiffErrorMin : Unit:bar
   // Signals[15].DiffErrorMin : Unit:bar
   // Signals[16].DiffErrorMin : Unit:bar
   // Signals[17].DiffErrorMin : Unit:bar
   // Signals[18].DiffErrorMin : Unit:mm/s
   // Signals[19].DiffErrorMin : Unit:mm/s
   // Signals[21].DiffErrorMin : Unit:°C
   // Signals[26].DiffErrorMin : Unit:°C
   // Signals[1].DiffWarnMax : Unit:W
   // Signals[3].DiffWarnMax : Unit:bar
   // Signals[4].DiffWarnMax : Unit:°C
   // Signals[5].DiffWarnMax : Unit:°C
   // Signals[6].DiffWarnMax : Unit:°C
   // Signals[7].DiffWarnMax : Unit:°C
   // Signals[8].DiffWarnMax : Unit:°C
   // Signals[9].DiffWarnMax : Unit:°C
   // Signals[10].DiffWarnMax : Unit:°C
   // Signals[13].DiffWarnMax : Unit:bar
   // Signals[14].DiffWarnMax : Unit:bar
   // Signals[15].DiffWarnMax : Unit:bar
   // Signals[16].DiffWarnMax : Unit:bar
   // Signals[17].DiffWarnMax : Unit:bar
   // Signals[18].DiffWarnMax : Unit:mm/s
   // Signals[19].DiffWarnMax : Unit:mm/s
   // Signals[21].DiffWarnMax : Unit:°C
   // Signals[26].DiffWarnMax : Unit:°C
   // Signals[1].DiffWarnMin : Unit:W
   // Signals[3].DiffWarnMin : Unit:bar
   // Signals[4].DiffWarnMin : Unit:°C
   // Signals[5].DiffWarnMin : Unit:°C
   // Signals[6].DiffWarnMin : Unit:°C
   // Signals[7].DiffWarnMin : Unit:°C
   // Signals[8].DiffWarnMin : Unit:°C
   // Signals[9].DiffWarnMin : Unit:°C
   // Signals[10].DiffWarnMin : Unit:°C
   // Signals[13].DiffWarnMin : Unit:bar
   // Signals[14].DiffWarnMin : Unit:bar
   // Signals[15].DiffWarnMin : Unit:bar
   // Signals[16].DiffWarnMin : Unit:bar
   // Signals[17].DiffWarnMin : Unit:bar
   // Signals[18].DiffWarnMin : Unit:mm/s
   // Signals[19].DiffWarnMin : Unit:mm/s
   // Signals[21].DiffWarnMin : Unit:°C
   // Signals[26].DiffWarnMin : Unit:°C
   // Signals[1].Offset : Unit:W
   // Signals[3].Offset : Unit:bar
   // Signals[4].Offset : Unit:°C
   // Signals[5].Offset : Unit:°C
   // Signals[6].Offset : Unit:°C
   // Signals[7].Offset : Unit:°C
   // Signals[8].Offset : Unit:°C
   // Signals[9].Offset : Unit:°C
   // Signals[10].Offset : Unit:°C
   // Signals[13].Offset : Unit:bar
   // Signals[14].Offset : Unit:bar
   // Signals[15].Offset : Unit:bar
   // Signals[16].Offset : Unit:bar
   // Signals[17].Offset : Unit:bar
   // Signals[18].Offset : Unit:mm/s
   // Signals[19].Offset : Unit:mm/s
   // Signals[21].Offset : Unit:°C
   // Signals[26].Offset : Unit:°C
   // Signals[1].Target : Unit:W
   // Signals[3].Target : Unit:bar
   // Signals[4].Target : Unit:°C
   // Signals[5].Target : Unit:°C
   // Signals[6].Target : Unit:°C
   // Signals[7].Target : Unit:°C
   // Signals[8].Target : Unit:°C
   // Signals[9].Target : Unit:°C
   // Signals[10].Target : Unit:°C
   // Signals[13].Target : Unit:bar
   // Signals[14].Target : Unit:bar
   // Signals[15].Target : Unit:bar
   // Signals[16].Target : Unit:bar
   // Signals[17].Target : Unit:bar
   // Signals[18].Target : Unit:mm/s
   // Signals[19].Target : Unit:mm/s
   // Signals[21].Target : Unit:°C
   // Signals[26].Target : Unit:°C
   // Signals[1].Value : Unit:W
   // Signals[3].Value : Unit:bar
   // Signals[4].Value : Unit:°C
   // Signals[5].Value : Unit:°C
   // Signals[6].Value : Unit:°C
   // Signals[7].Value : Unit:°C
   // Signals[8].Value : Unit:°C
   // Signals[9].Value : Unit:°C
   // Signals[10].Value : Unit:°C
   // Signals[13].Value : Unit:bar
   // Signals[14].Value : Unit:bar
   // Signals[15].Value : Unit:bar
   // Signals[16].Value : Unit:bar
   // Signals[17].Value : Unit:bar
   // Signals[18].Value : Unit:mm/s
   // Signals[19].Value : Unit:mm/s
   // Signals[21].Value : Unit:°C
   // Signals[26].Value : Unit:°C
END_DATA_BLOCK

DATA_BLOCK "DB_OPC_Components"   // DB118
{ S7_Optimized_Access := 'TRUE' }
// stored: MemoryReserve 100
   VAR
      Backwalls : Struct
         LoaderDrilled : Byte;
         LoaderUndrilled : Byte;
         Shuttle2Drilled : Byte;
         Shuttle2Undrilled : Byte;
         ShuttleDrilled : Byte;
         ShuttleUndrilled : Byte;
         WorkClamp : Byte;
      END_STRUCT;
      Parts : Struct
         LoaderDrilled : Byte;
         LoaderUndrilled : Byte;
         Shuttle2Drilled : Byte;
         Shuttle2Undrilled : Byte;
         ShuttleDrilled : Byte;
         ShuttleUndrilled : Byte;
         WorkClamp : Byte;
      END_STRUCT;
      Update : Byte;
   END_VAR
BEGIN
END_DATA_BLOCK

DATA_BLOCK "DB_NcVarSelect_R_Param"   // DB127
{ S7_Optimized_Access := 'TRUE' }
// stored: MemoryReserve 100
   VAR
      "$R[96]" { S7_SetPoint := 'True'} : "LBP_typeNCVariableTokenLReal";
      "$R[97]" { S7_SetPoint := 'True'} : "LBP_typeNCVariableTokenLReal";
      "$R[95]" { S7_SetPoint := 'True'} : "LBP_typeNCVariableTokenLReal";
      "$R[94]" { S7_SetPoint := 'True'} : SINU_typeNcVarTokenLReal;
   END_VAR
BEGIN
   "$R[96]".token.syntaxId := 16#82;
   "$R[96]".token.areaAndUnit := 16#41;
   "$R[96]".token.column := 16#1;
   "$R[96]".token.row := 16#61;
   "$R[96]".token.blockType := 16#15;
   "$R[96]".token.numberOfRows := 16#1;
   "$R[96]".token.dataTypeCode := 16#F;
   "$R[96]".token.length := 16#8;
   "$R[97]".token.syntaxId := 16#82;
   "$R[97]".token.areaAndUnit := 16#41;
   "$R[97]".token.column := 16#1;
   "$R[97]".token.row := 16#62;
   "$R[97]".token.blockType := 16#15;
   "$R[97]".token.numberOfRows := 16#1;
   "$R[97]".token.dataTypeCode := 16#F;
   "$R[97]".token.length := 16#8;
   "$R[95]".token.syntaxId := 16#82;
   "$R[95]".token.areaAndUnit := 16#41;
   "$R[95]".token.column := 16#1;
   "$R[95]".token.row := 16#60;
   "$R[95]".token.blockType := 16#15;
   "$R[95]".token.numberOfRows := 16#1;
   "$R[95]".token.dataTypeCode := 16#F;
   "$R[95]".token.length := 16#8;
   "$R[94]".token.syntaxId := 16#82;
   "$R[94]".token.areaAndUnit := 16#41;
   "$R[94]".token.column := 16#1;
   "$R[94]".token.row := 16#5F;
   "$R[94]".token.blockType := 16#15;
   "$R[94]".token.rowCount := 16#1;
   "$R[94]".token.dataType := 16#F;
   "$R[94]".token.length := 16#8;
END_DATA_BLOCK

DATA_BLOCK "DB_OPC_Laser"   // DB125
{ S7_Optimized_Access := 'TRUE' }
// stored: MemoryReserve 100
   VAR
      Scanner : Struct
         In : Struct
            CheckNumber : Byte;
            Ready : Bool;
            Status : DInt;
            StatusDescription : String;
         END_STRUCT;
         Out : Struct
            Parameters : Struct
               IsFirstJobOfPiece : Bool;
               StationNumber : Byte;
               HoleNumber : DInt;
               JobListName : String;
               JobName : String;
               MeasureZ : LReal;
            END_STRUCT;
            RequestJob : Bool;
            CheckNumber : Byte;
         END_STRUCT;
      END_STRUCT;
   END_VAR
BEGIN
END_DATA_BLOCK

DATA_BLOCK "R_Parameters"   // DB124
{ S7_Optimized_Access := 'TRUE' }
// stored: MemoryReserve 100
   VAR
      "$R[96]" { S7_SetPoint := 'True'} : SINU_typeNcVarTokenLReal;
      "$R[97]" { S7_SetPoint := 'True'} : SINU_typeNcVarTokenLReal;
      "$R[95]" { S7_SetPoint := 'True'} : SINU_typeNcVarTokenLReal;
      "$R[94]" { S7_SetPoint := 'True'} : SINU_typeNcVarTokenLReal;
   END_VAR
BEGIN
   "$R[96]".token.syntaxId := 16#82;
   "$R[96]".token.areaAndUnit := 16#41;
   "$R[96]".token.column := 16#1;
   "$R[96]".token.row := 16#61;
   "$R[96]".token.blockType := 16#15;
   "$R[96]".token.rowCount := 16#1;
   "$R[96]".token.dataType := 16#F;
   "$R[96]".token.length := 16#8;
   "$R[97]".token.syntaxId := 16#82;
   "$R[97]".token.areaAndUnit := 16#41;
   "$R[97]".token.column := 16#1;
   "$R[97]".token.row := 16#62;
   "$R[97]".token.blockType := 16#15;
   "$R[97]".token.rowCount := 16#1;
   "$R[97]".token.dataType := 16#F;
   "$R[97]".token.length := 16#8;
   "$R[95]".token.syntaxId := 16#82;
   "$R[95]".token.areaAndUnit := 16#41;
   "$R[95]".token.column := 16#1;
   "$R[95]".token.row := 16#60;
   "$R[95]".token.blockType := 16#15;
   "$R[95]".token.rowCount := 16#1;
   "$R[95]".token.dataType := 16#F;
   "$R[95]".token.length := 16#8;
   "$R[94]".token.syntaxId := 16#82;
   "$R[94]".token.areaAndUnit := 16#41;
   "$R[94]".token.column := 16#1;
   "$R[94]".token.row := 16#5F;
   "$R[94]".token.blockType := 16#15;
   "$R[94]".token.rowCount := 16#1;
   "$R[94]".token.dataType := 16#F;
   "$R[94]".token.length := 16#8;
END_DATA_BLOCK

DATA_BLOCK "DB_OPC_Recipe"   // DB134
{ S7_Optimized_Access := 'TRUE' }
// stored: MemoryReserve 100
   VAR RETAIN
      Current : Struct
         RecipeId : DInt;
         RecipeVersionGuid : String;
      END_STRUCT;
   END_VAR
   VAR
      Data : Struct
         LaserJobListName : String;
         RecipeId : DInt;
         RecipeName : String;
         RecipeVersionGuid : String;
         Station1 : Struct
            General : Struct
               Detections : Struct
                  WorkPart : Struct
                     Max : LReal;
                     Min : LReal;
                  END_STRUCT;
               END_STRUCT;
               GazPressure : Struct
                  WorkLaserDefault : LReal;
               END_STRUCT;
            END_STRUCT;
         END_STRUCT;
      END_STRUCT;
      TransferToPlc : Bool;
   END_VAR
BEGIN
END_DATA_BLOCK

DATA_BLOCK "DB_OPC_Maintenance"   // DB93
{ S7_Optimized_Access := 'TRUE' }
// stored: MemoryReserve 100
   VAR
      NumberOfTasks : Int := 16;
      Tasks : Array[0..100] of "UDT_OPC_Maintenance";
   END_VAR
BEGIN
END_DATA_BLOCK

DATA_BLOCK "LBP_CtrlEnergy"   // DB1000
TITLE = Ctrl-Energy
{ S7_Optimized_Access := 'FALSE'; DB_Accessible_From_OPC_UA := 'FALSE' }
AUTHOR : SINUMERIK
FAMILY : SINUMERIK_ONE
VERSION : 6.24
// Interface between user program and operating software, contains energy-saving profiles for Ctrl-Energy / Interface entre programme utilisateur et logiciel d'exploitation contient des profils d'économie d'énergie pour Ctrl-Energy
// stored: AutoNumber false, DBAccessibleFromOPCUA false, DBAccessibleFromWebserver false
   VAR RETAIN
      Profile : Array[1..8] of Struct
         ESaveOn { ExternalWritable := 'False'} : Bool;   // Activate energy-saving profile immediately / Activer immédiatement le profil d'économie d'énergie
         ReloadT2 { ExternalWritable := 'False'} : Bool;   // Reload Prewarning time (T2) / Recharger temps de préavis (T2)
         res0_2 { ExternalWritable := 'False'} : Bool;
         res0_3 { ExternalWritable := 'False'} : Bool;
         res0_4 { ExternalWritable := 'False'} : Bool;
         res0_5 { ExternalWritable := 'False'} : Bool;
         res0_6 { ExternalWritable := 'False'} : Bool;
         res0_7 { ExternalWritable := 'False'} : Bool;
         HmiESaveOn : Bool;   // HMI->PLC: Activate energy-saving profile immediately / IHM->AP : activer immédiatement le profil d'économie d'énergie
         res1_1 { ExternalWritable := 'False'} : Bool;
         res1_2 { ExternalWritable := 'False'} : Bool;
         res1_3 { ExternalWritable := 'False'} : Bool;
         res1_4 { ExternalWritable := 'False'} : Bool;
         res1_5 { ExternalWritable := 'False'} : Bool;
         res1_6 { ExternalWritable := 'False'} : Bool;
         res1_7 { ExternalWritable := 'False'} : Bool;
         MasterCompSig { ExternalWritable := 'False'} : Bool;   // Master computer signal / Signal ordinateur maître
         PlcUserSig { ExternalWritable := 'False'} : Bool;   // PLC user signal / AP signal utilisateur
         res2_2 { ExternalWritable := 'False'} : Bool;
         res2_3 { ExternalWritable := 'False'} : Bool;
         res2_4 { ExternalWritable := 'False'} : Bool;
         res2_5 { ExternalWritable := 'False'} : Bool;
         res2_6 { ExternalWritable := 'False'} : Bool;
         res2_7 { ExternalWritable := 'False'} : Bool;
         res3 { ExternalWritable := 'False'} : Byte;
         ESaveIsOn { ExternalWritable := 'False'} : Bool;   // Energy-saving state active / État économie d'énergie actif
         T1Expired { ExternalWritable := 'False'} : Bool;   // Activation time T1 expired / Temps d'activation T1 écoulé
         res4_2 { ExternalWritable := 'False'} : Bool;
         res4_3 { ExternalWritable := 'False'} : Bool;
         res4_4 { ExternalWritable := 'False'} : Bool;
         res4_5 { ExternalWritable := 'False'} : Bool;
         res4_6 { ExternalWritable := 'False'} : Bool;
         res4_7 { ExternalWritable := 'False'} : Bool;
         res5 { ExternalWritable := 'False'} : Byte;
         ActValT1 { ExternalWritable := 'False'} : Int;   // T1 current value / T1 valeur réelle
         ActValT2 { ExternalWritable := 'False'} : Int;   // T2 current value / T2 valeur réelle
         ESaveValid : Bool;   // HMI->PLC: Energy-saving profile valid / IHM->AP : profil d'économie d'énergie valide
         ESaveOff : Bool;   // HMI->PLC: Deactivate energy-saving profileblock energy-saving profile / IHM->AP : désactiver/bloquer le profil d'économie d'énergie
         res10_2 { ExternalWritable := 'False'} : Bool;
         res10_3 { ExternalWritable := 'False'} : Bool;
         res10_4 { ExternalWritable := 'False'} : Bool;
         res10_5 { ExternalWritable := 'False'} : Bool;
         res10_6 { ExternalWritable := 'False'} : Bool;
         res10_7 { ExternalWritable := 'False'} : Bool;
         CondOpPanel : Bool;   // HMI->PLC: Operator panel / IHM->AP : pupitre opérateur
         CondDataTransfer : Bool;   // HMI->PLC: Data transfer / IHM->AP : transmission de données
         CondWindowChange : Bool;   // HMI->PLC: Window change / IHM->AP : changement de fenêtre
         res11_3 { ExternalWritable := 'False'} : Bool;
         res11_4 { ExternalWritable := 'False'} : Bool;
         res11_5 { ExternalWritable := 'False'} : Bool;
         res11_6 { ExternalWritable := 'False'} : Bool;
         res11_7 { ExternalWritable := 'False'} : Bool;
         CondMCP : Bool;   // HMI->PLC: Machine control panel / IHM->AP : pupitre opérateur machine
         res12_1 { ExternalWritable := 'False'} : Bool;
         res12_2 { ExternalWritable := 'False'} : Bool;
         res12_3 { ExternalWritable := 'False'} : Bool;
         res12_4 { ExternalWritable := 'False'} : Bool;
         res12_5 { ExternalWritable := 'False'} : Bool;
         res12_6 { ExternalWritable := 'False'} : Bool;
         res12_7 { ExternalWritable := 'False'} : Bool;
         CondNcChan1 : Bool;   // HMI->PLC: NC channel 1 in reset / IHM->AP : canal CN 1 en Reset
         CondNcChan2 : Bool;   // HMI->PLC: NC channel 2 in reset / IHM->AP : canal CN 2 en Reset
         CondNcChan3 : Bool;   // HMI->PLC: NC channel 3 in reset / IHM->AP : canal CN 3 en Reset
         CondNcChan4 : Bool;   // HMI->PLC: NC channel 4 in reset / IHM->AP : canal CN 4 en Reset
         CondNcChan5 : Bool;   // HMI->PLC: NC channel 5 in reset / IHM->AP : canal CN 5 en Reset
         CondNcChan6 : Bool;   // HMI->PLC: NC channel 6 in reset / IHM->AP : canal CN 6 en Reset
         CondNcChan7 : Bool;   // HMI->PLC: NC channel 7 in reset / IHM->AP : canal CN 7 en Reset
         CondNcChan8 : Bool;   // HMI->PLC: NC channel 8 in reset / IHM->AP : canal CN 8 en Reset
         CondNcChan9 : Bool;   // HMI->PLC: NC channel 9 in reset / IHM->AP : canal CN 9 en Reset
         CondNcChan10 : Bool;   // HMI->PLC: NC channel 10 in reset / IHM->AP : canal CN 10 en Reset
         res14_2 { ExternalWritable := 'False'} : Bool;
         res14_3 { ExternalWritable := 'False'} : Bool;
         res14_4 { ExternalWritable := 'False'} : Bool;
         res14_5 { ExternalWritable := 'False'} : Bool;
         res14_6 { ExternalWritable := 'False'} : Bool;
         res14_7 { ExternalWritable := 'False'} : Bool;
         CondMasterCompSig : Bool;   // HMI->PLC: Master computer signal / IHM->AP : signal ordinateur maître
         CondPlcUserSig : Bool;   // HMI->PLC: PLC user signal / IHM->AP : signal utilisateur AP
         res15_2 { ExternalWritable := 'False'} : Bool;
         res15_3 { ExternalWritable := 'False'} : Bool;
         res15_4 { ExternalWritable := 'False'} : Bool;
         res15_5 { ExternalWritable := 'False'} : Bool;
         res15_6 { ExternalWritable := 'False'} : Bool;
         res15_7 { ExternalWritable := 'False'} : Bool;
         PresetT1 : Int;   // HMI->PLC: Activation time T1 / IHM->AP : temps d'activation T1
         PresetT2 : Int;   // HMI->PLC: Prewarning time T2 / IHM->AP : temps de préavis T2
      END_STRUCT;
   END_VAR
BEGIN
   // Profile[2].ESaveOn : Activate energy-saving profile immediately / Activer immédiatement le profil d'économie d'énergie
   // Profile[3].ESaveOn : Activate energy-saving profile immediately / Activer immédiatement le profil d'économie d'énergie
   // Profile[4].ESaveOn : Activate energy-saving profile immediately / Activer immédiatement le profil d'économie d'énergie
   // Profile[5].ESaveOn : Activate energy-saving profile immediately / Activer immédiatement le profil d'économie d'énergie
   // Profile[6].ESaveOn : Activate energy-saving profile immediately / Activer immédiatement le profil d'économie d'énergie
   // Profile[7].ESaveOn : Activate energy-saving profile immediately / Activer immédiatement le profil d'économie d'énergie
   // Profile[8].ESaveOn : Activate energy-saving profile immediately / Activer immédiatement le profil d'économie d'énergie
   // Profile[2].ReloadT2 : Reload Prewarning time (T2) / Recharger temps de préavis (T2)
   // Profile[3].ReloadT2 : Reload Prewarning time (T2) / Recharger temps de préavis (T2)
   // Profile[4].ReloadT2 : Reload Prewarning time (T2) / Recharger temps de préavis (T2)
   // Profile[5].ReloadT2 : Reload Prewarning time (T2) / Recharger temps de préavis (T2)
   // Profile[6].ReloadT2 : Reload Prewarning time (T2) / Recharger temps de préavis (T2)
   // Profile[7].ReloadT2 : Reload Prewarning time (T2) / Recharger temps de préavis (T2)
   // Profile[8].ReloadT2 : Reload Prewarning time (T2) / Recharger temps de préavis (T2)
   // Profile[2].HmiESaveOn : HMI->PLC: Activate energy-saving profile immediately / IHM->AP : activer immédiatement le profil d'économie d'énergie
   // Profile[3].HmiESaveOn : HMI->PLC: Activate energy-saving profile immediately / IHM->AP : activer immédiatement le profil d'économie d'énergie
   // Profile[4].HmiESaveOn : HMI->PLC: Activate energy-saving profile immediately / IHM->AP : activer immédiatement le profil d'économie d'énergie
   // Profile[5].HmiESaveOn : HMI->PLC: Activate energy-saving profile immediately / IHM->AP : activer immédiatement le profil d'économie d'énergie
   // Profile[6].HmiESaveOn : HMI->PLC: Activate energy-saving profile immediately / IHM->AP : activer immédiatement le profil d'économie d'énergie
   // Profile[7].HmiESaveOn : HMI->PLC: Activate energy-saving profile immediately / IHM->AP : activer immédiatement le profil d'économie d'énergie
   // Profile[8].HmiESaveOn : HMI->PLC: Activate energy-saving profile immediately / IHM->AP : activer immédiatement le profil d'économie d'énergie
   // Profile[2].MasterCompSig : Master computer signal / Signal ordinateur maître
   // Profile[3].MasterCompSig : Master computer signal / Signal ordinateur maître
   // Profile[4].MasterCompSig : Master computer signal / Signal ordinateur maître
   // Profile[5].MasterCompSig : Master computer signal / Signal ordinateur maître
   // Profile[6].MasterCompSig : Master computer signal / Signal ordinateur maître
   // Profile[7].MasterCompSig : Master computer signal / Signal ordinateur maître
   // Profile[8].MasterCompSig : Master computer signal / Signal ordinateur maître
   // Profile[2].PlcUserSig : PLC user signal / AP signal utilisateur
   // Profile[3].PlcUserSig : PLC user signal / AP signal utilisateur
   // Profile[4].PlcUserSig : PLC user signal / AP signal utilisateur
   // Profile[5].PlcUserSig : PLC user signal / AP signal utilisateur
   // Profile[6].PlcUserSig : PLC user signal / AP signal utilisateur
   // Profile[7].PlcUserSig : PLC user signal / AP signal utilisateur
   // Profile[8].PlcUserSig : PLC user signal / AP signal utilisateur
   // Profile[2].ESaveIsOn : Energy-saving state active / État économie d'énergie actif
   // Profile[3].ESaveIsOn : Energy-saving state active / État économie d'énergie actif
   // Profile[4].ESaveIsOn : Energy-saving state active / État économie d'énergie actif
   // Profile[5].ESaveIsOn : Energy-saving state active / État économie d'énergie actif
   // Profile[6].ESaveIsOn : Energy-saving state active / État économie d'énergie actif
   // Profile[7].ESaveIsOn : Energy-saving state active / État économie d'énergie actif
   // Profile[8].ESaveIsOn : Energy-saving state active / État économie d'énergie actif
   // Profile[2].T1Expired : Activation time T1 expired / Temps d'activation T1 écoulé
   // Profile[3].T1Expired : Activation time T1 expired / Temps d'activation T1 écoulé
   // Profile[4].T1Expired : Activation time T1 expired / Temps d'activation T1 écoulé
   // Profile[5].T1Expired : Activation time T1 expired / Temps d'activation T1 écoulé
   // Profile[6].T1Expired : Activation time T1 expired / Temps d'activation T1 écoulé
   // Profile[7].T1Expired : Activation time T1 expired / Temps d'activation T1 écoulé
   // Profile[8].T1Expired : Activation time T1 expired / Temps d'activation T1 écoulé
   // Profile[2].ActValT1 : T1 current value / T1 valeur réelle
   // Profile[3].ActValT1 : T1 current value / T1 valeur réelle
   // Profile[4].ActValT1 : T1 current value / T1 valeur réelle
   // Profile[5].ActValT1 : T1 current value / T1 valeur réelle
   // Profile[6].ActValT1 : T1 current value / T1 valeur réelle
   // Profile[7].ActValT1 : T1 current value / T1 valeur réelle
   // Profile[8].ActValT1 : T1 current value / T1 valeur réelle
   // Profile[2].ActValT2 : T2 current value / T2 valeur réelle
   // Profile[3].ActValT2 : T2 current value / T2 valeur réelle
   // Profile[4].ActValT2 : T2 current value / T2 valeur réelle
   // Profile[5].ActValT2 : T2 current value / T2 valeur réelle
   // Profile[6].ActValT2 : T2 current value / T2 valeur réelle
   // Profile[7].ActValT2 : T2 current value / T2 valeur réelle
   // Profile[8].ActValT2 : T2 current value / T2 valeur réelle
   Profile[1].ESaveValid := TRUE;
   Profile[2].ESaveValid := TRUE;   // HMI->PLC: Energy-saving profile valid / IHM->AP : profil d'économie d'énergie valide
   Profile[3].ESaveValid := TRUE;   // HMI->PLC: Energy-saving profile valid / IHM->AP : profil d'économie d'énergie valide
   // Profile[4].ESaveValid : HMI->PLC: Energy-saving profile valid / IHM->AP : profil d'économie d'énergie valide
   // Profile[5].ESaveValid : HMI->PLC: Energy-saving profile valid / IHM->AP : profil d'économie d'énergie valide
   // Profile[6].ESaveValid : HMI->PLC: Energy-saving profile valid / IHM->AP : profil d'économie d'énergie valide
   // Profile[7].ESaveValid : HMI->PLC: Energy-saving profile valid / IHM->AP : profil d'économie d'énergie valide
   // Profile[8].ESaveValid : HMI->PLC: Energy-saving profile valid / IHM->AP : profil d'économie d'énergie valide
   Profile[1].ESaveOff := TRUE;
   Profile[2].ESaveOff := TRUE;   // HMI->PLC: Deactivate energy-saving profileblock energy-saving profile / IHM->AP : désactiver/bloquer le profil d'économie d'énergie
   Profile[3].ESaveOff := TRUE;   // HMI->PLC: Deactivate energy-saving profileblock energy-saving profile / IHM->AP : désactiver/bloquer le profil d'économie d'énergie
   // Profile[4].ESaveOff : HMI->PLC: Deactivate energy-saving profileblock energy-saving profile / IHM->AP : désactiver/bloquer le profil d'économie d'énergie
   // Profile[5].ESaveOff : HMI->PLC: Deactivate energy-saving profileblock energy-saving profile / IHM->AP : désactiver/bloquer le profil d'économie d'énergie
   // Profile[6].ESaveOff : HMI->PLC: Deactivate energy-saving profileblock energy-saving profile / IHM->AP : désactiver/bloquer le profil d'économie d'énergie
   // Profile[7].ESaveOff : HMI->PLC: Deactivate energy-saving profileblock energy-saving profile / IHM->AP : désactiver/bloquer le profil d'économie d'énergie
   // Profile[8].ESaveOff : HMI->PLC: Deactivate energy-saving profileblock energy-saving profile / IHM->AP : désactiver/bloquer le profil d'économie d'énergie
   // Profile[2].CondOpPanel : HMI->PLC: Operator panel / IHM->AP : pupitre opérateur
   Profile[3].CondOpPanel := TRUE;   // HMI->PLC: Operator panel / IHM->AP : pupitre opérateur
   // Profile[4].CondOpPanel : HMI->PLC: Operator panel / IHM->AP : pupitre opérateur
   // Profile[5].CondOpPanel : HMI->PLC: Operator panel / IHM->AP : pupitre opérateur
   // Profile[6].CondOpPanel : HMI->PLC: Operator panel / IHM->AP : pupitre opérateur
   // Profile[7].CondOpPanel : HMI->PLC: Operator panel / IHM->AP : pupitre opérateur
   // Profile[8].CondOpPanel : HMI->PLC: Operator panel / IHM->AP : pupitre opérateur
   // Profile[2].CondDataTransfer : HMI->PLC: Data transfer / IHM->AP : transmission de données
   Profile[3].CondDataTransfer := TRUE;   // HMI->PLC: Data transfer / IHM->AP : transmission de données
   // Profile[4].CondDataTransfer : HMI->PLC: Data transfer / IHM->AP : transmission de données
   // Profile[5].CondDataTransfer : HMI->PLC: Data transfer / IHM->AP : transmission de données
   // Profile[6].CondDataTransfer : HMI->PLC: Data transfer / IHM->AP : transmission de données
   // Profile[7].CondDataTransfer : HMI->PLC: Data transfer / IHM->AP : transmission de données
   // Profile[8].CondDataTransfer : HMI->PLC: Data transfer / IHM->AP : transmission de données
   // Profile[2].CondWindowChange : HMI->PLC: Window change / IHM->AP : changement de fenêtre
   Profile[3].CondWindowChange := TRUE;   // HMI->PLC: Window change / IHM->AP : changement de fenêtre
   // Profile[4].CondWindowChange : HMI->PLC: Window change / IHM->AP : changement de fenêtre
   // Profile[5].CondWindowChange : HMI->PLC: Window change / IHM->AP : changement de fenêtre
   // Profile[6].CondWindowChange : HMI->PLC: Window change / IHM->AP : changement de fenêtre
   // Profile[7].CondWindowChange : HMI->PLC: Window change / IHM->AP : changement de fenêtre
   // Profile[8].CondWindowChange : HMI->PLC: Window change / IHM->AP : changement de fenêtre
   Profile[2].CondMCP := TRUE;   // HMI->PLC: Machine control panel / IHM->AP : pupitre opérateur machine
   Profile[3].CondMCP := TRUE;   // HMI->PLC: Machine control panel / IHM->AP : pupitre opérateur machine
   // Profile[4].CondMCP : HMI->PLC: Machine control panel / IHM->AP : pupitre opérateur machine
   // Profile[5].CondMCP : HMI->PLC: Machine control panel / IHM->AP : pupitre opérateur machine
   // Profile[6].CondMCP : HMI->PLC: Machine control panel / IHM->AP : pupitre opérateur machine
   // Profile[7].CondMCP : HMI->PLC: Machine control panel / IHM->AP : pupitre opérateur machine
   // Profile[8].CondMCP : HMI->PLC: Machine control panel / IHM->AP : pupitre opérateur machine
   Profile[1].CondNcChan1 := TRUE;
   Profile[2].CondNcChan1 := TRUE;   // HMI->PLC: NC channel 1 in reset / IHM->AP : canal CN 1 en Reset
   Profile[3].CondNcChan1 := TRUE;   // HMI->PLC: NC channel 1 in reset / IHM->AP : canal CN 1 en Reset
   // Profile[4].CondNcChan1 : HMI->PLC: NC channel 1 in reset / IHM->AP : canal CN 1 en Reset
   // Profile[5].CondNcChan1 : HMI->PLC: NC channel 1 in reset / IHM->AP : canal CN 1 en Reset
   // Profile[6].CondNcChan1 : HMI->PLC: NC channel 1 in reset / IHM->AP : canal CN 1 en Reset
   // Profile[7].CondNcChan1 : HMI->PLC: NC channel 1 in reset / IHM->AP : canal CN 1 en Reset
   // Profile[8].CondNcChan1 : HMI->PLC: NC channel 1 in reset / IHM->AP : canal CN 1 en Reset
   Profile[1].CondNcChan2 := TRUE;
   Profile[2].CondNcChan2 := TRUE;   // HMI->PLC: NC channel 2 in reset / IHM->AP : canal CN 2 en Reset
   Profile[3].CondNcChan2 := TRUE;   // HMI->PLC: NC channel 2 in reset / IHM->AP : canal CN 2 en Reset
   // Profile[4].CondNcChan2 : HMI->PLC: NC channel 2 in reset / IHM->AP : canal CN 2 en Reset
   // Profile[5].CondNcChan2 : HMI->PLC: NC channel 2 in reset / IHM->AP : canal CN 2 en Reset
   // Profile[6].CondNcChan2 : HMI->PLC: NC channel 2 in reset / IHM->AP : canal CN 2 en Reset
   // Profile[7].CondNcChan2 : HMI->PLC: NC channel 2 in reset / IHM->AP : canal CN 2 en Reset
   // Profile[8].CondNcChan2 : HMI->PLC: NC channel 2 in reset / IHM->AP : canal CN 2 en Reset
   Profile[1].CondNcChan3 := TRUE;
   Profile[2].CondNcChan3 := TRUE;   // HMI->PLC: NC channel 3 in reset / IHM->AP : canal CN 3 en Reset
   Profile[3].CondNcChan3 := TRUE;   // HMI->PLC: NC channel 3 in reset / IHM->AP : canal CN 3 en Reset
   // Profile[4].CondNcChan3 : HMI->PLC: NC channel 3 in reset / IHM->AP : canal CN 3 en Reset
   // Profile[5].CondNcChan3 : HMI->PLC: NC channel 3 in reset / IHM->AP : canal CN 3 en Reset
   // Profile[6].CondNcChan3 : HMI->PLC: NC channel 3 in reset / IHM->AP : canal CN 3 en Reset
   // Profile[7].CondNcChan3 : HMI->PLC: NC channel 3 in reset / IHM->AP : canal CN 3 en Reset
   // Profile[8].CondNcChan3 : HMI->PLC: NC channel 3 in reset / IHM->AP : canal CN 3 en Reset
   Profile[1].CondNcChan4 := TRUE;
   Profile[2].CondNcChan4 := TRUE;   // HMI->PLC: NC channel 4 in reset / IHM->AP : canal CN 4 en Reset
   Profile[3].CondNcChan4 := TRUE;   // HMI->PLC: NC channel 4 in reset / IHM->AP : canal CN 4 en Reset
   // Profile[4].CondNcChan4 : HMI->PLC: NC channel 4 in reset / IHM->AP : canal CN 4 en Reset
   // Profile[5].CondNcChan4 : HMI->PLC: NC channel 4 in reset / IHM->AP : canal CN 4 en Reset
   // Profile[6].CondNcChan4 : HMI->PLC: NC channel 4 in reset / IHM->AP : canal CN 4 en Reset
   // Profile[7].CondNcChan4 : HMI->PLC: NC channel 4 in reset / IHM->AP : canal CN 4 en Reset
   // Profile[8].CondNcChan4 : HMI->PLC: NC channel 4 in reset / IHM->AP : canal CN 4 en Reset
   Profile[1].CondNcChan5 := TRUE;
   Profile[2].CondNcChan5 := TRUE;   // HMI->PLC: NC channel 5 in reset / IHM->AP : canal CN 5 en Reset
   Profile[3].CondNcChan5 := TRUE;   // HMI->PLC: NC channel 5 in reset / IHM->AP : canal CN 5 en Reset
   // Profile[4].CondNcChan5 : HMI->PLC: NC channel 5 in reset / IHM->AP : canal CN 5 en Reset
   // Profile[5].CondNcChan5 : HMI->PLC: NC channel 5 in reset / IHM->AP : canal CN 5 en Reset
   // Profile[6].CondNcChan5 : HMI->PLC: NC channel 5 in reset / IHM->AP : canal CN 5 en Reset
   // Profile[7].CondNcChan5 : HMI->PLC: NC channel 5 in reset / IHM->AP : canal CN 5 en Reset
   // Profile[8].CondNcChan5 : HMI->PLC: NC channel 5 in reset / IHM->AP : canal CN 5 en Reset
   Profile[1].CondNcChan6 := TRUE;
   Profile[2].CondNcChan6 := TRUE;   // HMI->PLC: NC channel 6 in reset / IHM->AP : canal CN 6 en Reset
   Profile[3].CondNcChan6 := TRUE;   // HMI->PLC: NC channel 6 in reset / IHM->AP : canal CN 6 en Reset
   // Profile[4].CondNcChan6 : HMI->PLC: NC channel 6 in reset / IHM->AP : canal CN 6 en Reset
   // Profile[5].CondNcChan6 : HMI->PLC: NC channel 6 in reset / IHM->AP : canal CN 6 en Reset
   // Profile[6].CondNcChan6 : HMI->PLC: NC channel 6 in reset / IHM->AP : canal CN 6 en Reset
   // Profile[7].CondNcChan6 : HMI->PLC: NC channel 6 in reset / IHM->AP : canal CN 6 en Reset
   // Profile[8].CondNcChan6 : HMI->PLC: NC channel 6 in reset / IHM->AP : canal CN 6 en Reset
   Profile[1].CondNcChan7 := TRUE;
   Profile[2].CondNcChan7 := TRUE;   // HMI->PLC: NC channel 7 in reset / IHM->AP : canal CN 7 en Reset
   Profile[3].CondNcChan7 := TRUE;   // HMI->PLC: NC channel 7 in reset / IHM->AP : canal CN 7 en Reset
   // Profile[4].CondNcChan7 : HMI->PLC: NC channel 7 in reset / IHM->AP : canal CN 7 en Reset
   // Profile[5].CondNcChan7 : HMI->PLC: NC channel 7 in reset / IHM->AP : canal CN 7 en Reset
   // Profile[6].CondNcChan7 : HMI->PLC: NC channel 7 in reset / IHM->AP : canal CN 7 en Reset
   // Profile[7].CondNcChan7 : HMI->PLC: NC channel 7 in reset / IHM->AP : canal CN 7 en Reset
   // Profile[8].CondNcChan7 : HMI->PLC: NC channel 7 in reset / IHM->AP : canal CN 7 en Reset
   Profile[1].CondNcChan8 := TRUE;
   Profile[2].CondNcChan8 := TRUE;   // HMI->PLC: NC channel 8 in reset / IHM->AP : canal CN 8 en Reset
   Profile[3].CondNcChan8 := TRUE;   // HMI->PLC: NC channel 8 in reset / IHM->AP : canal CN 8 en Reset
   // Profile[4].CondNcChan8 : HMI->PLC: NC channel 8 in reset / IHM->AP : canal CN 8 en Reset
   // Profile[5].CondNcChan8 : HMI->PLC: NC channel 8 in reset / IHM->AP : canal CN 8 en Reset
   // Profile[6].CondNcChan8 : HMI->PLC: NC channel 8 in reset / IHM->AP : canal CN 8 en Reset
   // Profile[7].CondNcChan8 : HMI->PLC: NC channel 8 in reset / IHM->AP : canal CN 8 en Reset
   // Profile[8].CondNcChan8 : HMI->PLC: NC channel 8 in reset / IHM->AP : canal CN 8 en Reset
   Profile[1].CondNcChan9 := TRUE;
   Profile[2].CondNcChan9 := TRUE;   // HMI->PLC: NC channel 9 in reset / IHM->AP : canal CN 9 en Reset
   Profile[3].CondNcChan9 := TRUE;   // HMI->PLC: NC channel 9 in reset / IHM->AP : canal CN 9 en Reset
   // Profile[4].CondNcChan9 : HMI->PLC: NC channel 9 in reset / IHM->AP : canal CN 9 en Reset
   // Profile[5].CondNcChan9 : HMI->PLC: NC channel 9 in reset / IHM->AP : canal CN 9 en Reset
   // Profile[6].CondNcChan9 : HMI->PLC: NC channel 9 in reset / IHM->AP : canal CN 9 en Reset
   // Profile[7].CondNcChan9 : HMI->PLC: NC channel 9 in reset / IHM->AP : canal CN 9 en Reset
   // Profile[8].CondNcChan9 : HMI->PLC: NC channel 9 in reset / IHM->AP : canal CN 9 en Reset
   Profile[1].CondNcChan10 := TRUE;
   Profile[2].CondNcChan10 := TRUE;   // HMI->PLC: NC channel 10 in reset / IHM->AP : canal CN 10 en Reset
   Profile[3].CondNcChan10 := TRUE;   // HMI->PLC: NC channel 10 in reset / IHM->AP : canal CN 10 en Reset
   // Profile[4].CondNcChan10 : HMI->PLC: NC channel 10 in reset / IHM->AP : canal CN 10 en Reset
   // Profile[5].CondNcChan10 : HMI->PLC: NC channel 10 in reset / IHM->AP : canal CN 10 en Reset
   // Profile[6].CondNcChan10 : HMI->PLC: NC channel 10 in reset / IHM->AP : canal CN 10 en Reset
   // Profile[7].CondNcChan10 : HMI->PLC: NC channel 10 in reset / IHM->AP : canal CN 10 en Reset
   // Profile[8].CondNcChan10 : HMI->PLC: NC channel 10 in reset / IHM->AP : canal CN 10 en Reset
   // Profile[2].CondMasterCompSig : HMI->PLC: Master computer signal / IHM->AP : signal ordinateur maître
   // Profile[3].CondMasterCompSig : HMI->PLC: Master computer signal / IHM->AP : signal ordinateur maître
   // Profile[4].CondMasterCompSig : HMI->PLC: Master computer signal / IHM->AP : signal ordinateur maître
   // Profile[5].CondMasterCompSig : HMI->PLC: Master computer signal / IHM->AP : signal ordinateur maître
   // Profile[6].CondMasterCompSig : HMI->PLC: Master computer signal / IHM->AP : signal ordinateur maître
   // Profile[7].CondMasterCompSig : HMI->PLC: Master computer signal / IHM->AP : signal ordinateur maître
   // Profile[8].CondMasterCompSig : HMI->PLC: Master computer signal / IHM->AP : signal ordinateur maître
   Profile[1].CondPlcUserSig := TRUE;
   Profile[2].CondPlcUserSig := TRUE;   // HMI->PLC: PLC user signal / IHM->AP : signal utilisateur AP
   Profile[3].CondPlcUserSig := TRUE;   // HMI->PLC: PLC user signal / IHM->AP : signal utilisateur AP
   // Profile[4].CondPlcUserSig : HMI->PLC: PLC user signal / IHM->AP : signal utilisateur AP
   // Profile[5].CondPlcUserSig : HMI->PLC: PLC user signal / IHM->AP : signal utilisateur AP
   // Profile[6].CondPlcUserSig : HMI->PLC: PLC user signal / IHM->AP : signal utilisateur AP
   // Profile[7].CondPlcUserSig : HMI->PLC: PLC user signal / IHM->AP : signal utilisateur AP
   // Profile[8].CondPlcUserSig : HMI->PLC: PLC user signal / IHM->AP : signal utilisateur AP
   Profile[1].PresetT1 := 60;
   Profile[2].PresetT1 := 120;   // HMI->PLC: Activation time T1 / IHM->AP : temps d'activation T1
   Profile[3].PresetT1 := 600;   // HMI->PLC: Activation time T1 / IHM->AP : temps d'activation T1
   // Profile[4].PresetT1 : HMI->PLC: Activation time T1 / IHM->AP : temps d'activation T1
   // Profile[5].PresetT1 : HMI->PLC: Activation time T1 / IHM->AP : temps d'activation T1
   // Profile[6].PresetT1 : HMI->PLC: Activation time T1 / IHM->AP : temps d'activation T1
   // Profile[7].PresetT1 : HMI->PLC: Activation time T1 / IHM->AP : temps d'activation T1
   // Profile[8].PresetT1 : HMI->PLC: Activation time T1 / IHM->AP : temps d'activation T1
   Profile[1].PresetT2 := 120;
   Profile[2].PresetT2 := 300;   // HMI->PLC: Prewarning time T2 / IHM->AP : temps de préavis T2
   // Profile[3].PresetT2 : HMI->PLC: Prewarning time T2 / IHM->AP : temps de préavis T2
   // Profile[4].PresetT2 : HMI->PLC: Prewarning time T2 / IHM->AP : temps de préavis T2
   // Profile[5].PresetT2 : HMI->PLC: Prewarning time T2 / IHM->AP : temps de préavis T2
   // Profile[6].PresetT2 : HMI->PLC: Prewarning time T2 / IHM->AP : temps de préavis T2
   // Profile[7].PresetT2 : HMI->PLC: Prewarning time T2 / IHM->AP : temps de préavis T2
   // Profile[8].PresetT2 : HMI->PLC: Prewarning time T2 / IHM->AP : temps de préavis T2
END_DATA_BLOCK

DATA_BLOCK "LBP_MFuncDecListConfig"   // DB75
TITLE = M decoding acc. to list / Décodage M selon liste
{ S7_Optimized_Access := 'FALSE' }
AUTHOR : SINUMERIK
FAMILY : SINUMERIK_ONE
VERSION : 6.24
// Interface between user program and NCK, contains the configuration for the M functions to be decoded / Interface entre programme utilisateur et NCK contient la configuration des fonctions M à décoder.
// stored: AutoNumber false
   VAR RETAIN
      MSigGrp : Array[1..16] of Struct
         MExtAdr : Int;
         MFirstAdr : DInt;
         MLastAdr : DInt;
      END_STRUCT;
   END_VAR
BEGIN
   MSigGrp[1..16].MFirstAdr := DINT#0;
   MSigGrp[1..16].MLastAdr := DINT#0;
END_DATA_BLOCK

DATA_BLOCK "LBP_MFuncDecListSignals"   // DB76
TITLE = M decoding acc. to list / Décodage M selon liste
{ S7_Optimized_Access := 'FALSE' }
AUTHOR : SINUMERIK
FAMILY : SINUMERIK_ONE
VERSION : 6.24
// Interface between user program and NCK, contains the signal list for the request and acknowledgment of the M functions configured with LBP_MFuncDecListConfig [DB75] / Interface entre programme utilisateur et NCK contient la liste des signaux pour la demande et l'acquittement des fonctions M configurées avec LBP_MFuncDecListConfig [DB75]
// stored: AutoNumber false
   VAR
      MSigGrp1 : Struct
         MSig : Array[0..15] of Bool;
      END_STRUCT;
      MSigGrp2 : Struct
         MSig : Array[0..15] of Bool;
      END_STRUCT;
      MSigGrp3 : Struct
         MSig : Array[0..15] of Bool;
      END_STRUCT;
      MSigGrp4 : Struct
         MSig : Array[0..15] of Bool;
      END_STRUCT;
      MSigGrp5 : Struct
         MSig : Array[0..15] of Bool;
      END_STRUCT;
      MSigGrp6 : Struct
         MSig : Array[0..15] of Bool;
      END_STRUCT;
      MSigGrp7 : Struct
         MSig : Array[0..15] of Bool;
      END_STRUCT;
      MSigGrp8 : Struct
         MSig : Array[0..15] of Bool;
      END_STRUCT;
      MSigGrp9 : Struct
         MSig : Array[0..15] of Bool;
      END_STRUCT;
      MSigGrp10 : Struct
         MSig : Array[0..15] of Bool;
      END_STRUCT;
      MSigGrp11 : Struct
         MSig : Array[0..15] of Bool;
      END_STRUCT;
      MSigGrp12 : Struct
         MSig : Array[0..15] of Bool;
      END_STRUCT;
      MSigGrp13 : Struct
         MSig : Array[0..15] of Bool;
      END_STRUCT;
      MSigGrp14 : Struct
         MSig : Array[0..15] of Bool;
      END_STRUCT;
      MSigGrp15 : Struct
         MSig : Array[0..15] of Bool;
      END_STRUCT;
      MSigGrp16 : Struct
         MSig : Array[0..15] of Bool;
      END_STRUCT;
   END_VAR
BEGIN
END_DATA_BLOCK

DATA_BLOCK "LBP_PIServices"   // DB16
TITLE = PI Services / Services PI
// Interface for LBP_ReqPIService [FB7], contains definitions for all available PI services. / L'interface pour LBP_ReqPIService [FB7] contient des définitions pour tous les services PI disponibles.
   VAR
      SELECT : Struct
         PIName : String[10] := '_N_SELECT';
         p01 : Byte := BYTE#16#03;   // Area / Unit / Zone/unité
         p02 : Char := '2';   // Area identifier / Identificateur de zone
         p11 : Byte := BYTE#16#FD;   // Path name / Nom de chemin
         p12 : Byte := BYTE#16#13;   // Add string with arbitrary number of odd numbers / Ajouter une chaîne contenant un nombre quelconque de nombres impairs
         p21 : Byte := BYTE#16#FE;   // Program name / Nom de programme
         p22 : Byte := BYTE#16#13;   // Add string with arbitrary number of odd numbers / Ajouter une chaîne contenant un nombre quelconque de nombres impairs
      END_STRUCT;
      ASUP : Struct
         PIName : String[10] := '_N_ASUP__';
         p01 : Byte := BYTE#16#03;   // Area / Unit / Zone/unité
         p02 : Char := '2';   // Area identifier / Identificateur de zone
         p11 : Byte := BYTE#16#03;   // Interrupt number / Numéro d'interruption
         p12 : Byte := BYTE#16#05;   // Int from WORD specification / INT de spécification WORD
         p21 : Byte := BYTE#16#03;   // Priority / Priorité
         p22 : Byte := BYTE#16#05;   // Int from WORD specification / INT de spécification WORD
         p31 : Byte := BYTE#16#01;   // Liftfast
         p32 : Byte := BYTE#16#05;   // Int from WORD specification / INT de spécification WORD
         p41 : Byte := BYTE#16#01;   // Blocksync
         p42 : Byte := BYTE#16#05;   // Int from WORD specification / INT de spécification WORD
         p51 : Byte := BYTE#16#FD;   // Path name / Nom de chemin
         p52 : Byte := BYTE#16#13;   // Add string with arbitrary number of odd numbers / Ajouter une chaîne contenant un nombre quelconque de nombres impairs
         p61 : Byte := BYTE#16#FE;   // Program name / Nom de programme
         p62 : Byte := BYTE#16#13;   // Add string with arbitrary number of odd numbers / Ajouter une chaîne contenant un nombre quelconque de nombres impairs
      END_STRUCT;
      FINDBL : Struct
         PIName : String[10] := '_N_FINDBL';
         p01 : Byte := BYTE#16#03;   // Area / Unit / Zone/unité
         p02 : Char := '2';
         p11 : Byte := BYTE#16#01;   // Preprocessing mode / Mode de prétraitement
         p12 : Byte := BYTE#16#04;   // Word from WORD specification / Mot depuis spécification WORD
      END_STRUCT;
      SETUFR : Struct
         PIName : String[10] := '_N_SETUFR';
         p01 : Byte := BYTE#16#03;   // Area / Unit / Zone/unité
         p02 : Char := '2';
      END_STRUCT;
      CANCEL : Struct
         PIName : String[10] := '_N_CANCEL';
         p01 : Byte := BYTE#16#03;   // Area / Unit / Zone/unité
         p02 : Char := '0';
      END_STRUCT;
      DELETO : Struct
         PIName : String[10] := '_N_DELETO';
         p01 : Byte := BYTE#16#03;   // Area / Unit / Zone/unité
         p02 : Char := '4';
         p11 : Byte := BYTE#16#05;   // T number / Numéro d'outil
         p12 : Byte := BYTE#16#05;   // Int from WORD specification / INT de spécification WORD
      END_STRUCT;
      CREATO : Struct
         PIName : String[10] := '_N_CREATO';
         p01 : Byte := BYTE#16#03;   // Area / Unit / Zone/unité
         p02 : Char := '4';
         p11 : Byte := BYTE#16#05;   // T number / Numéro d'outil
         p12 : Byte := BYTE#16#05;   // Int from WORD specification / INT de spécification WORD
      END_STRUCT;
      CREACE : Struct
         PIName : String[10] := '_N_CREACE';
         p01 : Byte := BYTE#16#03;   // Area / Unit / Zone/unité
         p02 : Char := '4';
         p11 : Byte := BYTE#16#05;   // T number / Numéro d'outil
         p12 : Byte := BYTE#16#05;   // Int from WORD specification / INT de spécification WORD
      END_STRUCT;
      TMCRTO : Struct
         PIName : String[10] := '_N_TMCRTO';
         p01 : Byte := BYTE#16#03;   // Area / Unit / Zone/unité
         p02 : Char := '4';
         p11 : Byte := BYTE#16#20;   // Tool identifier, add blank / Identifiant d'outil, ajouter espace
         p12 : Byte := BYTE#16#13;   // String identifier! / Identifiant de chaîne.
         p21 : Byte := BYTE#16#05;   // T number / Numéro d'outil
         p22 : Byte := BYTE#16#05;   // Int from WORD specification / INT de spécification WORD
         p31 : Byte := BYTE#16#05;   // Duplo number / Numéro d'outil frère
         p32 : Byte := BYTE#16#05;   // Int from WORD specification / INT de spécification WORD
      END_STRUCT;
      TMFDPL : Struct
         PIName : String[10] := '_N_TMFDPL';
         p01 : Byte := BYTE#16#03;   // Area / Unit / Zone/unité
         p02 : Char := '4';
         p11 : Byte := BYTE#16#05;   // T number / Numéro d'outil
         p12 : Byte := BYTE#16#05;   // Int from WORD specification / INT de spécification WORD
         p21 : Byte := BYTE#16#05;   // Location number (target) / Numéro d'emplacement (cible)
         p22 : Byte := BYTE#16#05;   // Int from WORD specification / INT de spécification WORD
         p31 : Byte := BYTE#16#05;   // Magazine number (target) / Numéro de magasin (cible)
         p32 : Byte := BYTE#16#05;   // Int from WORD specification / INT de spécification WORD
         p41 : Byte := BYTE#16#05;   // Location number (reference) / Numéro d'emplacement (référence)
         p42 : Byte := BYTE#16#05;   // Int from WORD specification / INT de spécification WORD
         p51 : Byte := BYTE#16#05;   // Magazine number (reference) / ID Numéro de magasin (référence)
         p52 : Byte := BYTE#16#05;   // Int from WORD specification / INT de spécification WORD
      END_STRUCT;
      TMMVTL : Struct
         PIName : String[10] := '_N_TMMVTL';
         p01 : Byte := BYTE#16#03;   // Area / Unit / Zone/unité
         p02 : Char := '4';
         p11 : Byte := BYTE#16#05;   // T number / Numéro d'outil
         p12 : Byte := BYTE#16#05;   // Int from WORD specification / INT de spécification WORD
         p21 : Byte := BYTE#16#05;   // Location number (source) / Numéro d'emplacement (source)
         p22 : Byte := BYTE#16#05;   // Int from WORD specification / INT de spécification WORD
         p31 : Byte := BYTE#16#05;   // Magazine number (source) / Numéro de magasin (source)
         p32 : Byte := BYTE#16#05;   // Int from WORD specification / INT de spécification WORD
         p41 : Byte := BYTE#16#05;   // Location number (target) / Numéro d'emplacement (cible)
         p42 : Byte := BYTE#16#05;   // Int from WORD specification / INT de spécification WORD
         p51 : Byte := BYTE#16#05;   // Magazine number (target) / Numéro de magasin (cible)
         p52 : Byte := BYTE#16#05;   // Int from WORD specification / INT de spécification WORD
      END_STRUCT;
      TMPCIT : Struct
         PIName : String[10] := '_N_TMPCIT';
         p01 : Byte := BYTE#16#03;   // Area / Unit / Zone/unité
         p02 : Char := '4';
         p11 : Byte := BYTE#16#03;   // Spindle number / Numéro de broche
         p12 : Byte := BYTE#16#05;   // Int from WORD specification / INT de spécification WORD
         p21 : Byte := BYTE#16#05;   // Increment value / Incrément valeur
         p22 : Byte := BYTE#16#05;   // Int from WORD specification / INT de spécification WORD
      END_STRUCT;
      TMPOSM : Struct
         PIName : String[10] := '_N_TMPOSM';
         p01 : Byte := BYTE#16#03;   // Area / Unit / Zone/unité
         p02 : Char := '4';
         p11 : Byte := BYTE#16#05;   // T number / Numéro d'outil
         p12 : Byte := BYTE#16#05;   // Int from WORD specification / INT de spécification WORD
         p21 : Byte := BYTE#16#20;   // Tool identifier, add blank / Identificateur d'outil, ajouter espace
         p22 : Byte := BYTE#16#13;   // String identifier! / Identifiant de chaîne.
         p31 : Byte := BYTE#16#05;   // Duplo number / Numéro d'outil frère
         p32 : Byte := BYTE#16#05;   // Int from WORD specification / INT de spécification WORD
         p41 : Byte := BYTE#16#05;   // Location number (source) / Numéro d'emplacement (source)
         p42 : Byte := BYTE#16#05;   // Int from WORD specification / INT de spécification WORD
         p51 : Byte := BYTE#16#05;   // Magazine number (source) / Numéro de magasin (source)
         p52 : Byte := BYTE#16#05;   // Int from WORD specification / INT de spécification WORD
         p61 : Byte := BYTE#16#05;   // Location number (target) / Numéro d'emplacement (cible)
         p62 : Byte := BYTE#16#05;   // Int from WORD specification / INT de spécification WORD
         p71 : Byte := BYTE#16#05;   // Magazine number (target) / Numéro de magasin (cible)
         p72 : Byte := BYTE#16#05;   // Int from WORD specification / INT de spécification WORD
      END_STRUCT;
      DIGION : Struct
         PIName : String[10] := '_N_DIGION';
         p01 : Byte := BYTE#16#03;   // Area / Unit / Zone/unité
         p02 : Char := '2';
      END_STRUCT;
      DIGIOF : Struct
         PIName : String[10] := '_N_DIGIOF';
         p01 : Byte := BYTE#16#03;   // Area / Unit / Zone/unité
         p02 : Char := '2';
      END_STRUCT;
      CONFIG : Struct
         PIName : String[10] := '_N_CONFIG';
         p01 : Byte := BYTE#16#03;   // Area / Unit / Zone/unité
         p02 : Char := '0';
         p11 : Byte := BYTE#16#02;   // Classification
         p12 : Byte := BYTE#16#04;   // Int from WORD specification / INT de spécification WORD
      END_STRUCT;
      LOGIN : Struct
         PIName : String[10] := '_N_LOGIN_';
         p01 : Byte := BYTE#16#03;   // Area / Unit / Zone/unité
         p02 : Char := '0';
         p11 : Byte := BYTE#16#20;   // Password (8 to 32 characters) / Mot de passe (8 à 32 caractères)
         p12 : Byte := BYTE#16#13;   // String identifier! / Identifiant de chaîne.
      END_STRUCT;
      LOGOUT : Struct
         PIName : String[10] := '_N_LOGOUT';
         p01 : Byte := BYTE#16#03;   // Area / Unit / Zone/unité
         p02 : Char := '0';
      END_STRUCT;
      MMCSEM : Struct
         PIName : String[10] := '_N_MMCSEM';
         p01 : Byte := BYTE#16#03;   // Area / Unit / Zone/unité
         p02 : Char := '2';
         p11 : Byte := BYTE#16#03;   // Function number / Numéro de fonction
         p12 : Byte := BYTE#16#05;   // Int from WORD specification / INT de spécification WORD
         p21 : Byte := BYTE#16#01;   // Semaphore value / Valeur sémaphore
         p22 : Byte := BYTE#16#05;   // Int from WORD specification / INT de spécification WORD
      END_STRUCT;
      DELECE : Struct
         PIName : String[10] := '_N_DELECE';
         p01 : Byte := BYTE#16#03;   // Area / Unit / Zone/unité
         p02 : Char := '4';
         p11 : Byte := BYTE#16#05;   // T number / Numéro d'outil
         p12 : Byte := BYTE#16#05;   // Int from WORD specification / INT de spécification WORD
         p21 : Byte := BYTE#16#05;   // D number / Numéro D
         p22 : Byte := BYTE#16#05;   // Int from WORD specification / INT de spécification WORD
      END_STRUCT;
      CRCEDN : Struct
         PIName : String[10] := '_N_CRCEDN';
         p01 : Byte := BYTE#16#03;   // Area / Unit / Zone/unité
         p02 : Char := '4';
         p11 : Byte := BYTE#16#05;   // T number / Numéro d'outil
         p12 : Byte := BYTE#16#05;   // Int from WORD specification / INT de spécification WORD
         p21 : Byte := BYTE#16#05;   // D number / Numéro D
         p22 : Byte := BYTE#16#05;   // Int from WORD specification / INT de spécification WORD
      END_STRUCT;
      TSEARC : Struct
         PIName : String[10] := '_N_TSEARC';
         p01 : Byte := BYTE#16#03;   // Area / Unit / Zone/unité
         p02 : Char := '4';
         p11 : Byte := BYTE#16#05;   // from: Magazine number / de : numéro de magasin
         p12 : Byte := BYTE#16#05;   // Int from WORD specification / INT de spécification WORD
         p21 : Byte := BYTE#16#05;   // from: Location number / de : numéro d'emplacement
         p22 : Byte := BYTE#16#05;   // Int from WORD specification / INT de spécification WORD
         p31 : Byte := BYTE#16#05;   // up to: Magazine number / à : numéro de magasin
         p32 : Byte := BYTE#16#05;   // Int from WORD specification / INT de spécification WORD
         p41 : Byte := BYTE#16#05;   // up to: Location number / à : numéro d'emplacement
         p42 : Byte := BYTE#16#05;   // Int from WORD specification / INT de spécification WORD
         p51 : Byte := BYTE#16#05;   // Number of reference magazine / Numéro du magasin de référence
         p52 : Byte := BYTE#16#05;   // Int from WORD specification / INT de spécification WORD
         p61 : Byte := BYTE#16#05;   // Number of reference location / Numéro de l'emplacement de référence
         p62 : Byte := BYTE#16#05;   // Int from WORD specification / INT de spécification WORD
         p71 : Byte := BYTE#16#01;   // Search direction / Sens de recherche
         p72 : Byte := BYTE#16#05;   // Int from WORD specification / INT de spécification WORD
         p81 : Byte := BYTE#16#01;   // Tool properties / Caractéristiques de l'outil
         p82 : Byte := BYTE#16#05;   // Int from WORD specification / INT de spécification WORD
      END_STRUCT;
      TMFPBP : Struct
         PIName : String[10] := '_N_TMFPBP';
         p01 : Byte := BYTE#16#03;   // Area / Unit / Zone/unité
         p02 : Char := '4';
         p11 : Byte := BYTE#16#05;   // from: Magazine number / de : numéro de magasin
         p12 : Byte := BYTE#16#05;   // Int from WORD specification / INT de spécification WORD
         p21 : Byte := BYTE#16#05;   // from: Location number / de : numéro d'emplacement
         p22 : Byte := BYTE#16#05;   // Int from WORD specification / INT de spécification WORD
         p31 : Byte := BYTE#16#05;   // up to: Magazine number / à : numéro de magasin
         p32 : Byte := BYTE#16#05;   // Int from WORD specification / INT de spécification WORD
         p41 : Byte := BYTE#16#05;   // up to: Location number / à : numéro d'emplacement
         p42 : Byte := BYTE#16#05;   // Int from WORD specification / INT de spécification WORD
         p51 : Byte := BYTE#16#05;   // Number of reference magazine / Numéro du magasin de référence
         p52 : Byte := BYTE#16#05;   // Int from WORD specification / INT de spécification WORD
         p61 : Byte := BYTE#16#05;   // Number of reference location / Numéro de l'emplacement de référence
         p62 : Byte := BYTE#16#05;   // Int from WORD specification / INT de spécification WORD
         p71 : Byte := BYTE#16#05;   // Number of locations to the left / Nombre d'emplacements vers la gauche
         p72 : Byte := BYTE#16#05;   // Int from WORD specification / INT de spécification WORD
         p81 : Byte := BYTE#16#05;   // Number of locations to the right / Nombre d'emplacements vers la droite
         p82 : Byte := BYTE#16#05;   // Int from WORD specification / INT de spécification WORD
         p91 { ExternalVisible := 'False'} : Byte := BYTE#16#05;   // Number of locations above / Nombre d'emplacements vers le haut
         p92 : Byte := BYTE#16#05;   // Int from WORD specification / INT de spécification WORD
         pa1 : Byte := BYTE#16#05;   // Number of locations below / Nombre d'emplacements vers le bas
         pa2 : Byte := BYTE#16#05;   // Int from WORD specification / INT de spécification WORD
         pb1 : Byte := BYTE#16#05;   // Location type index / Type d'emplacement Indice
         pb2 : Byte := BYTE#16#05;   // Int from WORD specification / INT de spécification WORD
         pc1 : Byte := BYTE#16#05;   // Search direction / Sens de recherche
         pc2 : Byte := BYTE#16#05;   // Int from WORD specification / INT de spécification WORD
      END_STRUCT;
      NCRES : Struct
         PIName : String[10] := '_N_IBN_SS';
         p01 : Byte := BYTE#16#03;   // Area / Unit / Zone/unité
         p02 : Char := 'K';
         p11 : Byte := BYTE#16#01;   // Classification
         p12 : Byte := BYTE#16#04;   // WORD specification / Spécification WORD
      END_STRUCT;
      TMRASS : Struct
         PIName : String[10] := '_N_TMRASS';
         p01 : Byte := BYTE#16#03;   // Area / Unit / Zone/unité
         p02 : Char := '4';
      END_STRUCT;
      TRESMO : Struct
         PIName : String[10] := '_N_TRESMO';
         p01 : Byte := BYTE#16#03;   // Area / Unit / Zone/unité
         p02 : Char := '4';
         p11 : Byte := BYTE#16#05;   // Tool number / Numéro d'outil
         p12 : Byte := BYTE#16#05;   // Int from WORD specification / INT de spécification WORD
         p21 : Byte := BYTE#16#05;   // D number / Numéro D
         p22 : Byte := BYTE#16#05;   // Int from WORD specification / INT de spécification WORD
         p31 : Byte := BYTE#16#05;   // Monitoring type / Type de surveillance
         p32 : Byte := BYTE#16#05;   // Int from WORD specification / INT de spécification WORD
      END_STRUCT;
      TMGETT : Struct
         PIName : String[10] := '_N_TMGETT';
         p01 : Byte := BYTE#16#03;   // Area / Unit / Zone/unité
         p02 : Char := '4';
         p11 : Byte := BYTE#16#20;   // Tool identifier, add blank / Identifiant d'outil, ajouter espace
         p12 : Byte := BYTE#16#13;   // String identifier! / Identifiant de chaîne.
         p21 : Byte := BYTE#16#05;   // Duplo number / Numéro d'outil frère
         p22 : Byte := BYTE#16#05;   // Int from WORD specification / INT de spécification WORD
      END_STRUCT;
      SETUDT : Struct
         PIName : String[10] := '_N_SETUDT';
         p01 : Byte := BYTE#16#03;   // Area / Unit / Zone/unité
         p02 : Char := '2';
         p11 : Byte := BYTE#16#03;   // UserDataType
         p12 : Byte := BYTE#16#04;   // WORD specification / Spécification WORD
         p21 : Byte := BYTE#16#05;   // ind1
         p22 : Byte := BYTE#16#04;   // WORD specification / Spécification WORD
         p31 : Byte := BYTE#16#05;   // ind2
         p32 : Byte := BYTE#16#04;   // WORD specification / Spécification WORD
      END_STRUCT;
      TMCRMT : Struct
         PIName : String[10] := '_N_TMCRMT';
         p01 : Byte := BYTE#16#03;   // Area / Unit / Zone/unité
         p02 : Char := '4';
         p11 : Byte := BYTE#16#20;   // Multitool identifier, insert blanks / Identifiant Multitool, ajouter espace
         p12 : Byte := BYTE#16#13;   // String identifier! / Identifiant de chaîne.
         p21 : Byte := BYTE#16#05;   // Reserved / Réservé
         p22 : Byte := BYTE#16#05;   // Int from WORD specification / INT de spécification WORD
         p31 : Byte := BYTE#16#05;   // Multitool number / Numéro Multitool
         p32 : Byte := BYTE#16#05;   // Int from WORD specification / INT de spécification WORD
         p41 : Byte := BYTE#16#03;   // Number of Multitool locations / Nombre d'emplacements Multitool
         p42 : Byte := BYTE#16#05;   // Int from WORD specification / INT de spécification WORD
         p51 : Byte := BYTE#16#01;   // Type of distance coding / Type de codage de distance
         p52 : Byte := BYTE#16#05;   // Int from WORD specification / INT de spécification WORD
      END_STRUCT;
      TMDLMT : Struct
         PIName : String[10] := '_N_TMDLMT';
         p01 : Byte := BYTE#16#03;   // Area / Unit / Zone/unité
         p02 : Char := '4';
         p11 : Byte := BYTE#16#20;   // Multitool identifier, insert blanks / Identifiant Multitool, ajouter espace
         p12 : Byte := BYTE#16#13;   // String identifier! / Identifiant de chaîne.
         p21 : Byte := BYTE#16#05;   // Reserved / Réservé
         p22 : Byte := BYTE#16#05;   // Int from WORD specification / INT de spécification WORD
         p31 : Byte := BYTE#16#05;   // Multitool number / Numéro Multitool
         p32 : Byte := BYTE#16#05;   // Int from WORD specification / INT de spécification WORD
         p41 : Byte := BYTE#16#01;   // Delete included tools / Supprimer les outils contenus
         p42 : Byte := BYTE#16#05;   // Int from WORD specification / INT de spécification WORD
      END_STRUCT;
      POSMT : Struct
         PIName : String[10] := '_N_POSMT_';
         p01 : Byte := BYTE#16#03;   // Area / Unit / Zone/unité
         p02 : Char := '4';
         p11 : Byte := BYTE#16#03;   // Number of toolholder / Numéro du porte-outil
         p12 : Byte := BYTE#16#05;   // Int from WORD specification / INT de spécification WORD
         p21 : Byte := BYTE#16#05;   // Tool number / Numéro d'outil
         p22 : Byte := BYTE#16#05;   // Int from WORD specification / INT de spécification WORD
         p31 : Byte := BYTE#16#20;   // Tool number, add blank / Identificateur d'outil, ajouter espace
         p32 : Byte := BYTE#16#13;   // String identifier! / Identifiant de chaîne.
         p41 : Byte := BYTE#16#05;   // Duplo number / Numéro d'outil frère
         p42 : Byte := BYTE#16#05;   // Int from WORD specification / INT de spécification WORD
         p51 : Byte := BYTE#16#03;   // Multitool place number / Numéro d'emplacement Multitool
         p52 : Byte := BYTE#16#05;   // Int from WORD specification / INT de spécification WORD
      END_STRUCT;
      FDPLMT : Struct
         PIName : String[10] := '_N_FDPLMT';
         p01 : Byte := BYTE#16#03;   // Area / Unit / Zone/unité
         p02 : Char := '4';
         p11 : Byte := BYTE#16#05;   // Tool number / Numéro d'outil
         p12 : Byte := BYTE#16#05;   // Int from WORD specification / INT de spécification WORD
         p21 : Byte := BYTE#16#20;   // Tool number, add blank / Identificateur d'outil, ajouter espace
         p22 : Byte := BYTE#16#13;   // String identifier! / Identifiant de chaîne.
         p31 : Byte := BYTE#16#05;   // Duplo number / Numéro d'outil frère
         p32 : Byte := BYTE#16#05;   // Int from WORD specification / INT de spécification WORD
         p41 : Byte := BYTE#16#05;   // Multitool number / Numéro Multitool
         p42 : Byte := BYTE#16#05;   // Int from WORD specification / INT de spécification WORD
         p51 : Byte := BYTE#16#03;   // Multitool place number / Numéro d'emplacement Multitool
         p52 : Byte := BYTE#16#05;   // Int from WORD specification / INT de spécification WORD
      END_STRUCT;
      RETRAC : Struct
         PIName : String[10] := '_N_RETRAC';
         p01 : Byte := BYTE#16#03;   // Area / Unit / Zone/unité
         p02 : Char := '2';
         p11 : Byte := BYTE#16#03;   // Geometry axis / Axe géométrique
         p12 : Byte := BYTE#16#04;   // WORD specification / Spécification WORD
         p21 : Byte := BYTE#16#05;   // Parameter2 / Paramètre2
         p22 : Byte := BYTE#16#04;   // WORD specification / Spécification WORD
      END_STRUCT;
   END_VAR
BEGIN
END_DATA_BLOCK

